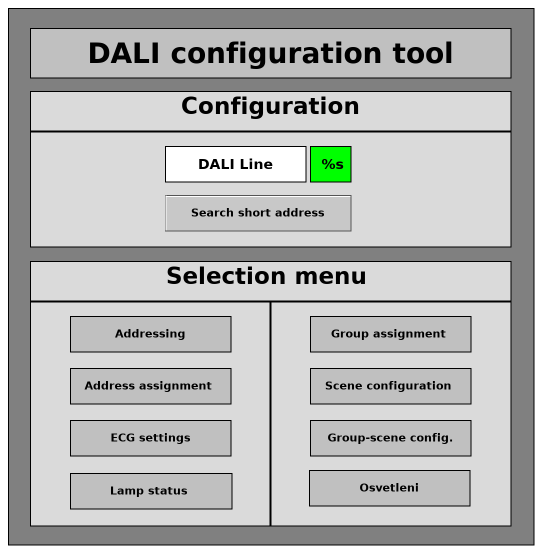
rectangle at (171,91)-(652,247): text "Configuration"
rectangle at (171,261)-(652,526): text "Selection menu"
rectangle at (171,28)-(652,78): text "DALI configuration tool"
rectangle at (211,316)-(372,352): text "Addressing"; opens Addressing
rectangle at (211,368)-(372,404): text "Address assignment"; opens Sort_short_address
rectangle at (451,316)-(612,352): text "Group assignment"; opens group_assignment
rectangle at (451,368)-(612,404): text "Scene configuration"; opens Scene_configuration
rectangle at (211,420)-(372,456): text "ECG settings"; opens ECG_settings
rectangle at (451,420)-(612,456): text "Group-scene config."; opens GroupSceneConfiguration
rectangle at (306,146)-(447,182): text "DALI Line"
button at (306,195)-(492,231): text "Search short address"; taps DALI_Config.SucheKurzadr; tooltip Clicking the button "Search Short Address" will start the search for available short addresses.
rectangle at (451,146)-(492,182): text "%s"; shows DALI_Config.Dali_Linie; alarm colour if DALI_Config.keineJobliste; tooltip Select DALI Line (1 - 5); editable
rectangle at (211,473)-(373,509): text "Lamp status"; opens Lamp_status
rectangle at (450,470)-(611,506): text "Osvetleni"; opens PLC_VISU
4 more shapes without text or variables
*)

(* Visualisation DALI_cfg
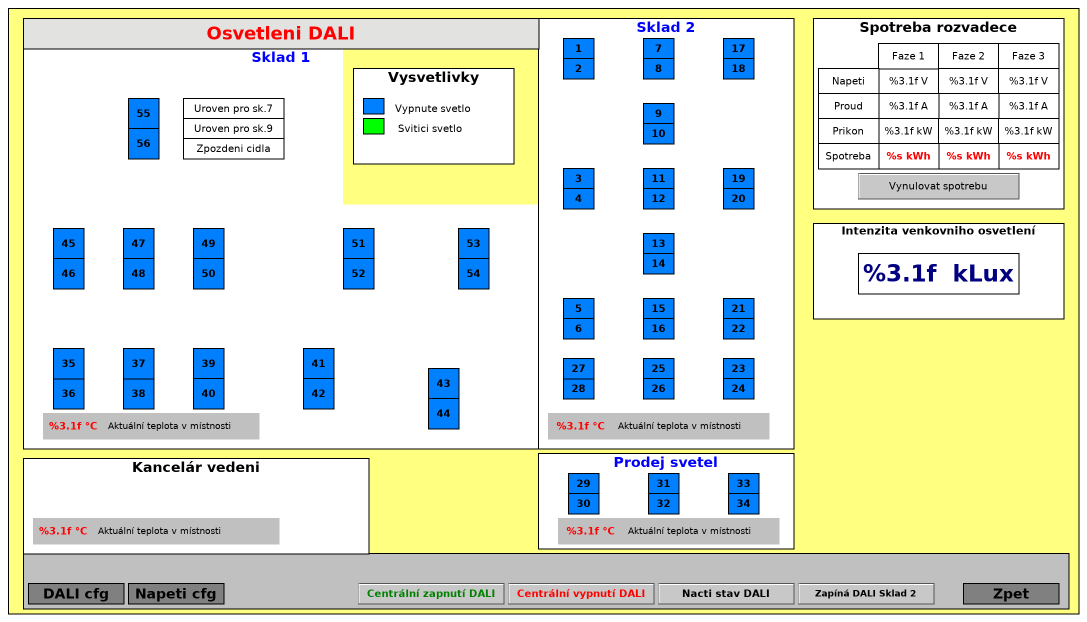
rectangle at (30,50)-(546,451): text "Sklad 1"
rounded rectangle at (360,70)-(521,166): text "Vysvetlivky"
rectangle at (545,455)-(801,551): text "Prodej svetel"; opens prodej_svetel
rectangle at (545,20)-(801,451): text "Sklad 2"; opens prodej_svetel
rectangle at (570,40)-(601,61): text "1"; alarm colour if DALI_Config.Kurzadr[1]
rectangle at (570,40)-(601,61): text "1"; invisible if not DALI_Config.Kurzadr[1]; alarm colour if DALI_Config.LampeEin[1]
rectangle at (570,60)-(601,81): text "2"; alarm colour if DALI_Config.Kurzadr[2]
rectangle at (570,60)-(601,81): text "2"; invisible if not DALI_Config.Kurzadr[2]; alarm colour if DALI_Config.LampeEin[2]
rectangle at (570,170)-(601,191): text "3"; alarm colour if DALI_Config.Kurzadr[3]
rectangle at (570,170)-(601,191): text "3"; invisible if not DALI_Config.Kurzadr[3]; alarm colour if DALI_Config.LampeEin[3]
rectangle at (570,190)-(601,211): text "4"; alarm colour if DALI_Config.Kurzadr[4]
rectangle at (570,190)-(601,211): text "4"; invisible if not DALI_Config.Kurzadr[4]; alarm colour if DALI_Config.LampeEin[4]
rectangle at (570,300)-(601,321): text "5"; alarm colour if DALI_Config.Kurzadr[5]
rectangle at (570,300)-(601,321): text "5"; invisible if not DALI_Config.Kurzadr[5]; alarm colour if DALI_Config.LampeEin[5]
rectangle at (570,320)-(601,341): text "6"; alarm colour if DALI_Config.Kurzadr[6]
rectangle at (570,320)-(601,341): text "6"; invisible if not DALI_Config.Kurzadr[6]; alarm colour if DALI_Config.LampeEin[6]
rectangle at (650,40)-(681,61): text "7"; alarm colour if DALI_Config.Kurzadr[7]
rectangle at (650,40)-(681,61): text "7"; invisible if not DALI_Config.Kurzadr[7]; alarm colour if DALI_Config.LampeEin[7]
rectangle at (650,60)-(681,81): text "8"; alarm colour if DALI_Config.Kurzadr[8]
rectangle at (650,60)-(681,81): text "8"; invisible if not DALI_Config.Kurzadr[8]; alarm colour if DALI_Config.LampeEin[8]
rectangle at (650,105)-(681,126): text "9"; alarm colour if DALI_Config.Kurzadr[9]
rectangle at (650,105)-(681,126): text "9"; invisible if not DALI_Config.Kurzadr[9]; alarm colour if DALI_Config.LampeEin[9]
rectangle at (650,125)-(681,146): text "10"; alarm colour if DALI_Config.Kurzadr[10]
rectangle at (650,125)-(681,146): text "10"; invisible if not DALI_Config.Kurzadr[10]; alarm colour if DALI_Config.LampeEin[10]
rectangle at (650,170)-(681,191): text "11"; alarm colour if DALI_Config.Kurzadr[11]
rectangle at (650,170)-(681,191): text "11"; invisible if not DALI_Config.Kurzadr[11]; alarm colour if DALI_Config.LampeEin[11]
rectangle at (650,190)-(681,211): text "12"; alarm colour if DALI_Config.Kurzadr[12]
rectangle at (650,190)-(681,211): text "12"; invisible if not DALI_Config.Kurzadr[12]; alarm colour if DALI_Config.LampeEin[12]
rectangle at (650,235)-(681,256): text "13"; alarm colour if DALI_Config.Kurzadr[13]
rectangle at (650,235)-(681,256): text "13"; invisible if not DALI_Config.Kurzadr[13]; alarm colour if DALI_Config.LampeEin[13]
rectangle at (650,255)-(681,276): text "14"; alarm colour if DALI_Config.Kurzadr[14]
rectangle at (650,255)-(681,276): text "14"; invisible if not DALI_Config.Kurzadr[14]; alarm colour if DALI_Config.LampeEin[14]
rectangle at (650,300)-(681,321): text "15"; alarm colour if DALI_Config.Kurzadr[15]
rectangle at (650,300)-(681,321): text "15"; invisible if not DALI_Config.Kurzadr[15]; alarm colour if DALI_Config.LampeEin[15]
rectangle at (650,320)-(681,341): text "16"; alarm colour if DALI_Config.Kurzadr[16]
rectangle at (650,320)-(681,341): text "16"; invisible if not DALI_Config.Kurzadr[16]; alarm colour if DALI_Config.LampeEin[16]
rectangle at (730,40)-(761,61): text "17"; alarm colour if DALI_Config.Kurzadr[17]
rectangle at (730,40)-(761,61): text "17"; invisible if not DALI_Config.Kurzadr[17]; alarm colour if DALI_Config.LampeEin[17]
rectangle at (730,170)-(761,191): text "19"; alarm colour if DALI_Config.Kurzadr[19]
rectangle at (730,170)-(761,191): text "19"; invisible if not DALI_Config.Kurzadr[19]; alarm colour if DALI_Config.LampeEin[19]
rectangle at (730,60)-(761,81): text "18"; alarm colour if DALI_Config.Kurzadr[18]
rectangle at (730,60)-(761,81): text "18"; invisible if not DALI_Config.Kurzadr[18]; alarm colour if DALI_Config.LampeEin[18]
rectangle at (730,190)-(761,211): text "20"; alarm colour if DALI_Config.Kurzadr[20]
rectangle at (730,190)-(761,211): text "20"; invisible if not DALI_Config.Kurzadr[20]; alarm colour if DALI_Config.LampeEin[20]
rectangle at (730,300)-(761,321): text "21"; alarm colour if DALI_Config.Kurzadr[21]
rectangle at (730,300)-(761,321): text "21"; invisible if not DALI_Config.Kurzadr[21]; alarm colour if DALI_Config.LampeEin[21]
rectangle at (730,320)-(761,341): text "22"; alarm colour if DALI_Config.Kurzadr[22]
rectangle at (730,320)-(761,341): text "22"; invisible if not DALI_Config.Kurzadr[22]; alarm colour if DALI_Config.LampeEin[22]
rectangle at (730,360)-(761,381): text "23"; alarm colour if DALI_Config.Kurzadr[23]
rectangle at (730,360)-(761,381): text "23"; invisible if not DALI_Config.Kurzadr[23]; alarm colour if DALI_Config.LampeEin[23]
rectangle at (730,380)-(761,401): text "24"; alarm colour if DALI_Config.Kurzadr[24]
rectangle at (730,380)-(761,401): text "24"; invisible if not DALI_Config.Kurzadr[24]; alarm colour if DALI_Config.LampeEin[24]
rectangle at (650,360)-(681,381): text "25"; alarm colour if DALI_Config.Kurzadr[25]
rectangle at (650,360)-(681,381): text "25"; invisible if not DALI_Config.Kurzadr[25]; alarm colour if DALI_Config.LampeEin[25]
rectangle at (575,475)-(606,496): text "29"; alarm colour if DALI_Config.Kurzadr[29]
rectangle at (575,475)-(606,496): text "29"; invisible if not DALI_Config.Kurzadr[29]; alarm colour if DALI_Config.LampeEin[29]
rectangle at (570,380)-(601,401): text "28"; alarm colour if DALI_Config.Kurzadr[28]
rectangle at (570,380)-(601,401): text "28"; invisible if not DALI_Config.Kurzadr[28]; alarm colour if DALI_Config.LampeEin[28]
rectangle at (570,360)-(601,381): text "27"; alarm colour if DALI_Config.Kurzadr[27]
rectangle at (570,360)-(601,381): text "27"; invisible if not DALI_Config.Kurzadr[27]; alarm colour if DALI_Config.LampeEin[27]
rectangle at (650,380)-(681,401): text "26"; alarm colour if DALI_Config.Kurzadr[26]
rectangle at (650,380)-(681,401): text "26"; invisible if not DALI_Config.Kurzadr[26]; alarm colour if DALI_Config.LampeEin[26]
rectangle at (575,495)-(606,516): text "30"; alarm colour if DALI_Config.Kurzadr[30]
rectangle at (575,495)-(606,516): text "30"; invisible if not DALI_Config.Kurzadr[30]; alarm colour if DALI_Config.LampeEin[30]
rectangle at (655,475)-(686,496): text "31"; alarm colour if DALI_Config.Kurzadr[31]
rectangle at (655,475)-(686,496): text "31"; invisible if not DALI_Config.Kurzadr[31]; alarm colour if DALI_Config.LampeEin[31]
rectangle at (655,495)-(686,516): text "32"; alarm colour if DALI_Config.Kurzadr[32]
rectangle at (655,495)-(686,516): text "32"; invisible if not DALI_Config.Kurzadr[32]; alarm colour if DALI_Config.LampeEin[32]
rectangle at (735,475)-(766,496): text "33"; alarm colour if DALI_Config.Kurzadr[33]
rectangle at (735,475)-(766,496): text "33"; invisible if not DALI_Config.Kurzadr[33]; alarm colour if DALI_Config.LampeEin[33]
rectangle at (735,495)-(766,516): text "34"; alarm colour if DALI_Config.Kurzadr[34]
rectangle at (735,495)-(766,516): text "34"; invisible if not DALI_Config.Kurzadr[34]; alarm colour if DALI_Config.LampeEin[34]
rectangle at (60,380)-(91,411): text "36"; alarm colour if DALI_Config.Kurzadr[36]
rectangle at (60,380)-(91,411): text "36"; invisible if not DALI_Config.Kurzadr[36]; alarm colour if DALI_Config.LampeEin[36]
rectangle at (130,380)-(161,411): text "38"; alarm colour if DALI_Config.Kurzadr[38]
rectangle at (130,380)-(161,411): text "38"; invisible if not DALI_Config.Kurzadr[38]; alarm colour if DALI_Config.LampeEin[38]
rectangle at (200,350)-(231,381): text "39"; alarm colour if DALI_Config.Kurzadr[39]
rectangle at (200,350)-(231,381): text "39"; invisible if not DALI_Config.Kurzadr[39]; alarm colour if DALI_Config.LampeEin[39]
rectangle at (130,350)-(161,381): text "37"; alarm colour if DALI_Config.Kurzadr[37]
rectangle at (130,350)-(161,381): text "37"; invisible if not DALI_Config.Kurzadr[37]; alarm colour if DALI_Config.LampeEin[37]
rectangle at (60,350)-(91,381): text "35"; alarm colour if DALI_Config.Kurzadr[35]
rectangle at (60,350)-(91,381): text "35"; invisible if not DALI_Config.Kurzadr[35]; alarm colour if DALI_Config.LampeEin[35]
rectangle at (310,350)-(341,381): text "41"; alarm colour if DALI_Config.Kurzadr[41]
rectangle at (310,350)-(341,381): text "41"; invisible if not DALI_Config.Kurzadr[41]; alarm colour if DALI_Config.LampeEin[41]
rectangle at (310,380)-(341,411): text "42"; alarm colour if DALI_Config.Kurzadr[42]
rectangle at (310,380)-(341,411): text "42"; invisible if not DALI_Config.Kurzadr[42]; alarm colour if DALI_Config.LampeEin[42]
rectangle at (200,380)-(231,411): text "40"; alarm colour if DALI_Config.Kurzadr[40]
rectangle at (200,380)-(231,411): text "40"; invisible if not DALI_Config.Kurzadr[40]; alarm colour if DALI_Config.LampeEin[40]
rectangle at (435,370)-(466,401): text "43"; alarm colour if DALI_Config.Kurzadr[43]
rectangle at (435,370)-(466,401): text "43"; invisible if not DALI_Config.Kurzadr[43]; alarm colour if DALI_Config.LampeEin[43]
rectangle at (435,400)-(466,431): text "44"; alarm colour if DALI_Config.Kurzadr[44]
rectangle at (435,400)-(466,431): text "44"; invisible if not DALI_Config.Kurzadr[44]; alarm colour if DALI_Config.LampeEin[44]
rectangle at (60,230)-(91,261): text "45"; alarm colour if DALI_Config.Kurzadr[45]
rectangle at (60,230)-(91,261): text "45"; invisible if not DALI_Config.Kurzadr[45]; alarm colour if DALI_Config.LampeEin[45]
rectangle at (60,260)-(91,291): text "46"; alarm colour if DALI_Config.Kurzadr[46]
rectangle at (60,260)-(91,291): text "46"; invisible if not DALI_Config.Kurzadr[46]; alarm colour if DALI_Config.LampeEin[46]
rectangle at (130,230)-(161,261): text "47"; alarm colour if DALI_Config.Kurzadr[47]
rectangle at (130,230)-(161,261): text "47"; invisible if not DALI_Config.Kurzadr[47]; alarm colour if DALI_Config.LampeEin[47]
rectangle at (130,260)-(161,291): text "48"; alarm colour if DALI_Config.Kurzadr[48]
rectangle at (130,260)-(161,291): text "48"; invisible if not DALI_Config.Kurzadr[48]; alarm colour if DALI_Config.LampeEin[48]
rectangle at (200,230)-(231,261): text "49"; alarm colour if DALI_Config.Kurzadr[49]
rectangle at (200,230)-(231,261): text "49"; invisible if not DALI_Config.Kurzadr[49]; alarm colour if DALI_Config.LampeEin[49]
rectangle at (200,260)-(231,291): text "50"; alarm colour if DALI_Config.Kurzadr[50]
rectangle at (200,260)-(231,291): text "50"; invisible if not DALI_Config.Kurzadr[50]; alarm colour if DALI_Config.LampeEin[50]
rectangle at (350,230)-(381,261): text "51"; alarm colour if DALI_Config.Kurzadr[51]
rectangle at (350,230)-(381,261): text "51"; invisible if not DALI_Config.Kurzadr[51]; alarm colour if DALI_Config.LampeEin[51]
rectangle at (350,260)-(381,291): text "52"; alarm colour if DALI_Config.Kurzadr[52]
rectangle at (350,260)-(381,291): text "52"; invisible if not DALI_Config.Kurzadr[52]; alarm colour if DALI_Config.LampeEin[52]
rectangle at (465,230)-(496,261): text "53"; alarm colour if DALI_Config.Kurzadr[53]
rectangle at (465,230)-(496,261): text "53"; invisible if not DALI_Config.Kurzadr[53]; alarm colour if DALI_Config.LampeEin[53]
rectangle at (465,260)-(496,291): text "54"; alarm colour if DALI_Config.Kurzadr[54]
rectangle at (465,260)-(496,291): text "54"; invisible if not DALI_Config.Kurzadr[54]; alarm colour if DALI_Config.LampeEin[54]
rectangle at (135,100)-(166,131): text "55"; alarm colour if DALI_Config.Kurzadr[55]
rectangle at (135,100)-(166,131): text "55"; invisible if not DALI_Config.Kurzadr[55]; alarm colour if DALI_Config.LampeEin[55]
rectangle at (135,130)-(166,161): text "56"; alarm colour if DALI_Config.Kurzadr[56]
rectangle at (135,130)-(166,161): text "56"; invisible if not DALI_Config.Kurzadr[56]; alarm colour if DALI_Config.LampeEin[56]
rectangle at (30,20)-(546,51): text "Osvetleni DALI"
button at (665,585)-(801,606): text "Nacti stav DALI"; taps DALI_Config.Status; tooltip Kliknutim nactete status svetel. (sviti, nesviti, vadna).
rectangle at (400,100)-(516,121): text "Vypnute svetlo"
rectangle at (400,120)-(536,141): text "Svitici svetlo"
rectangle at (565,520)-(631,546): text "%3.1f °C"; shows .Teplota_2/10.0
rectangle at (630,520)-(786,546): text "Aktuální teplota v místnosti"
rectangle at (620,415)-(776,441): text "Aktuální teplota v místnosti"
rectangle at (110,415)-(266,441): text "Aktuální teplota v místnosti"
rectangle at (555,415)-(621,441): text "%3.1f °C"; shows .Teplota_1/10.0
rectangle at (50,415)-(111,441): text "%3.1f °C"; shows .Teplota_3/10.0
button at (365,585)-(511,606): text "Centrální zapnutí DALI"; taps DALI_Config.Ein; tooltip Vsechny DALI svetla zapni
button at (515,585)-(661,606): text "Centrální vypnutí DALI"; taps DALI_Config.Aus; tooltip Vsechny DALI svetla vypni
rounded rectangle at (820,20)-(1071,211): text "Spotreba rozvadece"
rectangle at (885,70)-(946,96): text "%3.1f V"; shows TriFaze.arNapeti[1]
rectangle at (885,45)-(946,71): text "Faze 1"
rectangle at (945,45)-(1006,71): text "Faze 2"
rectangle at (1005,45)-(1066,71): text "Faze 3"
rectangle at (945,70)-(1006,96): text "%3.1f V"; shows TriFaze.arNapeti[2]
rectangle at (1005,70)-(1066,96): text "%3.1f V"; shows TriFaze.arNapeti[3]
rectangle at (1005,95)-(1066,121): text "%3.1f A"; shows TriFaze.arProud[3]
rectangle at (945,95)-(1006,121): text "%3.1f A"; shows TriFaze.arProud[2]
rectangle at (885,95)-(946,121): text "%3.1f A"; shows TriFaze.arProud[1]
rectangle at (885,120)-(946,146): text "%3.1f kW"; shows TriFaze.arVykon[1]
rectangle at (945,120)-(1006,146): text "%3.1f kW"; shows TriFaze.arVykon[2]
rectangle at (1005,120)-(1066,146): text "%3.1f kW"; shows TriFaze.arVykon[3]
rectangle at (1005,145)-(1066,171): text "%s kWh"; shows TriFaze.adwSpotreba[3]
rectangle at (945,145)-(1006,171): text "%s kWh"; shows TriFaze.adwSpotreba[2]
rectangle at (885,145)-(946,171): text "%s kWh"; shows TriFaze.adwSpotreba[1]
button at (865,175)-(1026,201): text "Vynulovat spotrebu"; taps TriFaze.SmazL1
rounded rectangle at (820,225)-(1071,321): text "Intenzita venkovniho osvetlení"; opens lux
rectangle at (865,255)-(1026,296): text "%3.1f  kLux"; shows .Analog_1/3276.4*2
rectangle at (825,70)-(886,96): text "Napeti"
rectangle at (825,95)-(886,121): text "Proud"
rectangle at (825,120)-(886,146): text "Prikon"
rectangle at (825,145)-(886,171): text "Spotreba"
rectangle at (30,460)-(376,556): text "Kancelár vedeni"
rectangle at (100,520)-(286,546): text "Aktuální teplota v místnosti"
rectangle at (40,520)-(101,546): text "%3.1f °C"; shows .Teplota_4/10.0
rectangle at (970,585)-(1066,606): text "Zpet"; opens PLC_VISU; tooltip Na úvodní stranu
rectangle at (135,585)-(231,606): text "Napeti cfg"; opens Visualizace; tooltip Back to home page
button at (805,585)-(941,606): text "Zapíná DALI Sklad 2"; taps .TL01s; tooltip 1x zapne/vypne, 2x zapne skupinu 2, 3x zapne vše
rectangle at (35,585)-(131,606): text "DALI cfg"; opens DALI; tooltip Back to home page
rectangle at (190,100)-(291,121): text "Uroven pro sk.7"
rectangle at (190,120)-(291,141): text "Uroven pro sk.9"
rectangle at (190,140)-(291,161): text "Zpozdeni cidla"
6 more shapes without text or variables
3 elements of other kinds (tables, trends, ...) not read
*)

(* Visualisation ECG_settings
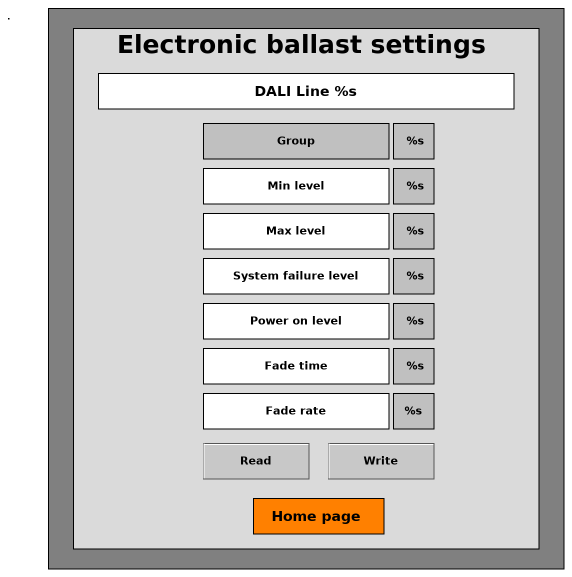
rectangle at (150,40)-(616,561): text "Electronic ballast settings"
rectangle at (280,225)-(466,261): text "Max level"
rectangle at (280,180)-(466,216): text "Min level"
rectangle at (280,270)-(466,306): text "System failure level"
rectangle at (280,315)-(466,351): text "Power on level"
rectangle at (280,360)-(466,396): text "Fade time"
rectangle at (280,405)-(466,441): text "Fade rate"
rectangle at (280,135)-(466,171): text "Short address"; invisible if DALI_Config.Kurzadr_Gruppe; toggles DALI_Config.Kurzadr_Gruppe
rectangle at (280,135)-(466,171): text "Group"; invisible if not DALI_Config.Kurzadr_Gruppe; toggles DALI_Config.Kurzadr_Gruppe; tooltip Selection group or short address
rectangle at (470,135)-(511,171): text "%s"; shows DALI_Config.Adresse; tooltip Enter group (1-16) or short address (1 - 64); editable
rounded rectangle at (330,510)-(461,546): text "Home page"; opens DALI; tooltip Back to home page
rectangle at (470,180)-(511,216): text "%s"; shows DALI_Config.MinLevel; tooltip Minimal brightness level in percent. Min level has to be smaller than max level.; editable
rectangle at (470,225)-(511,261): text "%s"; shows DALI_Config.MaxLevel; tooltip Maximum brightness level in percent; editable
rectangle at (470,270)-(511,306): text "%s"; shows DALI_Config.SystemFailure; tooltip Brightness level in percent in case of a system failure. The value 101 means "MASK".; editable
rectangle at (470,315)-(511,351): text "%s"; shows DALI_Config.PowerOn; tooltip Brightness level in percent if the ECGs are powered on.; editable
rectangle at (470,360)-(511,396): text "%s"; shows DALI_Config.Konfig[4]; tooltip Enter the fade time (0 - 15); editable
rectangle at (470,405)-(511,441): text "%s"; shows DALI_Config.Konfig[5]; tooltip Enter the fade rate (1 -15); editable
button at (280,455)-(386,491): text "Read"; taps DALI_Config.Lese; tooltip If you click the button "Read", the settings of the ECG will be read. Group queries are not possible.
button at (405,455)-(511,491): text "Write"; taps DALI_Config.Schreib; tooltip If you click the button "Write", the new settings will be written into the ECG.
rounded rectangle at (175,85)-(591,121): text "DALI Line %s"; shows DALI_Config.bDali_Linie; tooltip You can change the DALI Line only on the home page.
2 more shapes without text or variables
*)

(* Visualisation Group_assignment
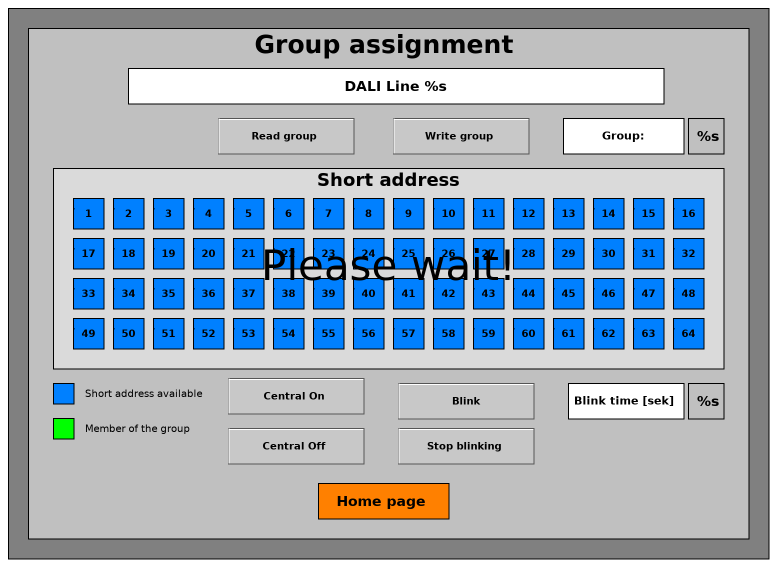
rectangle at (40,40)-(761,551): text "Group assignment"
rounded rectangle at (330,495)-(461,531): text "Home page"; opens DALI; tooltip Back to home page
rectangle at (65,180)-(736,381): text "Short address"
rectangle at (85,210)-(116,241): text "1"; alarm colour if DALI_Config.Kurzadr[1]
rectangle at (85,210)-(116,241): text "1"; invisible if not DALI_Config.Kurzadr[1]; alarm colour if DALI_Config.Gruppenadr[1]; toggles DALI_Config.Gruppenadr[1]
rectangle at (125,210)-(156,241): text "2"; alarm colour if DALI_Config.Kurzadr[2]
rectangle at (125,210)-(156,241): text "2"; invisible if not DALI_Config.Kurzadr[2]; alarm colour if DALI_Config.Gruppenadr[2]; toggles DALI_Config.Gruppenadr[2]
rectangle at (165,210)-(196,241): text "3"; alarm colour if DALI_Config.Kurzadr[3]
rectangle at (165,210)-(196,241): text "3"; invisible if not DALI_Config.Kurzadr[3]; alarm colour if DALI_Config.Gruppenadr[3]; toggles DALI_Config.Gruppenadr[3]
rectangle at (205,210)-(236,241): text "4"; alarm colour if DALI_Config.Kurzadr[4]
rectangle at (205,210)-(236,241): text "4"; invisible if not DALI_Config.Kurzadr[4]; alarm colour if DALI_Config.Gruppenadr[4]; toggles DALI_Config.Gruppenadr[4]
rectangle at (245,210)-(276,241): text "5"; alarm colour if DALI_Config.Kurzadr[5]
rectangle at (245,210)-(276,241): text "5"; invisible if not DALI_Config.Kurzadr[5]; alarm colour if DALI_Config.Gruppenadr[5]; toggles DALI_Config.Gruppenadr[5]
rectangle at (285,210)-(316,241): text "6"; alarm colour if DALI_Config.Kurzadr[6]
rectangle at (285,210)-(316,241): text "6"; invisible if not DALI_Config.Kurzadr[6]; alarm colour if DALI_Config.Gruppenadr[6]; toggles DALI_Config.Gruppenadr[6]
rectangle at (325,210)-(356,241): text "7"; alarm colour if DALI_Config.Kurzadr[7]
rectangle at (325,210)-(356,241): text "7"; invisible if not DALI_Config.Kurzadr[7]; alarm colour if DALI_Config.Gruppenadr[7]; toggles DALI_Config.Gruppenadr[7]
rectangle at (365,210)-(396,241): text "8"; alarm colour if DALI_Config.Kurzadr[8]
rectangle at (365,210)-(396,241): text "8"; invisible if not DALI_Config.Kurzadr[8]; alarm colour if DALI_Config.Gruppenadr[8]; toggles DALI_Config.Gruppenadr[8]
rectangle at (405,210)-(436,241): text "9"; alarm colour if DALI_Config.Kurzadr[9]
rectangle at (405,210)-(436,241): text "9"; invisible if not DALI_Config.Kurzadr[9]; alarm colour if DALI_Config.Gruppenadr[9]; toggles DALI_Config.Gruppenadr[9]
rectangle at (445,210)-(476,241): text "10"; alarm colour if DALI_Config.Kurzadr[10]
rectangle at (445,210)-(476,241): text "10"; invisible if not DALI_Config.Kurzadr[10]; alarm colour if DALI_Config.Gruppenadr[10]; toggles DALI_Config.Gruppenadr[10]
rectangle at (485,210)-(516,241): text "11"; alarm colour if DALI_Config.Kurzadr[11]
rectangle at (485,210)-(516,241): text "11"; invisible if not DALI_Config.Kurzadr[11]; alarm colour if DALI_Config.Gruppenadr[11]; toggles DALI_Config.Gruppenadr[11]
rectangle at (525,210)-(556,241): text "12"; alarm colour if DALI_Config.Kurzadr[12]
rectangle at (525,210)-(556,241): text "12"; invisible if not DALI_Config.Kurzadr[12]; alarm colour if DALI_Config.Gruppenadr[12]; toggles DALI_Config.Gruppenadr[12]
rectangle at (565,210)-(596,241): text "13"; alarm colour if DALI_Config.Kurzadr[13]
rectangle at (565,210)-(596,241): text "13"; invisible if not DALI_Config.Kurzadr[13]; alarm colour if DALI_Config.Gruppenadr[13]; toggles DALI_Config.Gruppenadr[13]
rectangle at (605,210)-(636,241): text "14"; alarm colour if DALI_Config.Kurzadr[14]
rectangle at (605,210)-(636,241): text "14"; invisible if not DALI_Config.Kurzadr[14]; alarm colour if DALI_Config.Gruppenadr[14]; toggles DALI_Config.Gruppenadr[14]
rectangle at (645,210)-(676,241): text "15"; alarm colour if DALI_Config.Kurzadr[15]
rectangle at (645,210)-(676,241): text "15"; invisible if not DALI_Config.Kurzadr[15]; alarm colour if DALI_Config.Gruppenadr[15]; toggles DALI_Config.Gruppenadr[15]
rectangle at (685,210)-(716,241): text "16"; alarm colour if DALI_Config.Kurzadr[16]
rectangle at (685,210)-(716,241): text "16"; invisible if not DALI_Config.Kurzadr[16]; alarm colour if DALI_Config.Gruppenadr[16]; toggles DALI_Config.Gruppenadr[16]
button at (405,130)-(541,166): text "Write group"; taps DALI_Config.Gruppenkonfiguration; tooltip If you click the button "Write Group", the marked short addresses will be saved as a group.
rectangle at (575,130)-(696,166): text "Group:"
rectangle at (700,130)-(736,166): text "%s"; shows DALI_Config.Gruppe; tooltip Enter the number of the group (1 - 16); editable
button at (410,395)-(546,431): text "Blink"; taps DALI_Config.BlinkenGruppe; tooltip If you click the button "Blink", the selected ECG will blink as long as defined by the "Blink Time" parameter.
button at (410,440)-(546,476): text "Stop blinking"; taps DALI_Config.xBlinken_Aus; tooltip If you click the button "Stop blinking", the blinking of the ECG will stop immediately.
button at (230,130)-(366,166): text "Read group"; taps DALI_Config.GruppeLesen; tooltip If you click the button "Read Group", the short addresses that belong to the group will be displayed.
rectangle at (95,395)-(226,416): text "Short address available"
rectangle at (95,430)-(246,451): text "Member of the group"
rounded rectangle at (140,80)-(676,116): text "DALI Line %s"; shows DALI_Config.bDali_Linie; tooltip You can change the DALI Line only on the home page.
rectangle at (85,250)-(116,281): text "17"; alarm colour if DALI_Config.Kurzadr[17]
rectangle at (85,250)-(116,281): text "17"; invisible if not DALI_Config.Kurzadr[17]; alarm colour if DALI_Config.Gruppenadr[17]; toggles DALI_Config.Gruppenadr[17]
rectangle at (125,250)-(156,281): text "18"; alarm colour if DALI_Config.Kurzadr[18]
rectangle at (125,250)-(156,281): text "18"; invisible if not DALI_Config.Kurzadr[18]; alarm colour if DALI_Config.Gruppenadr[18]; toggles DALI_Config.Gruppenadr[18]
rectangle at (165,250)-(196,281): text "19"; alarm colour if DALI_Config.Kurzadr[19]
rectangle at (165,250)-(196,281): text "19"; invisible if not DALI_Config.Kurzadr[19]; alarm colour if DALI_Config.Gruppenadr[19]; toggles DALI_Config.Gruppenadr[19]
rectangle at (205,250)-(236,281): text "20"; alarm colour if DALI_Config.Kurzadr[20]
rectangle at (205,250)-(236,281): text "20"; invisible if not DALI_Config.Kurzadr[20]; alarm colour if DALI_Config.Gruppenadr[20]; toggles DALI_Config.Gruppenadr[20]
rectangle at (245,250)-(276,281): text "21"; alarm colour if DALI_Config.Kurzadr[21]
rectangle at (245,250)-(276,281): text "21"; invisible if not DALI_Config.Kurzadr[21]; alarm colour if DALI_Config.Gruppenadr[21]; toggles DALI_Config.Gruppenadr[21]
rectangle at (285,250)-(316,281): text "22"; alarm colour if DALI_Config.Kurzadr[22]
rectangle at (285,250)-(316,281): text "22"; invisible if not DALI_Config.Kurzadr[22]; alarm colour if DALI_Config.Gruppenadr[22]; toggles DALI_Config.Gruppenadr[22]
rectangle at (325,250)-(356,281): text "23"; alarm colour if DALI_Config.Kurzadr[23]
rectangle at (325,250)-(356,281): text "23"; invisible if not DALI_Config.Kurzadr[23]; alarm colour if DALI_Config.Gruppenadr[23]; toggles DALI_Config.Gruppenadr[23]
rectangle at (365,250)-(396,281): text "24"; alarm colour if DALI_Config.Kurzadr[24]
rectangle at (365,250)-(396,281): text "24"; invisible if not DALI_Config.Kurzadr[24]; alarm colour if DALI_Config.Gruppenadr[24]; toggles DALI_Config.Gruppenadr[24]
rectangle at (405,250)-(436,281): text "25"; alarm colour if DALI_Config.Kurzadr[25]
rectangle at (405,250)-(436,281): text "25"; invisible if not DALI_Config.Kurzadr[25]; alarm colour if DALI_Config.Gruppenadr[25]; toggles DALI_Config.Gruppenadr[25]
rectangle at (445,250)-(476,281): text "26"; alarm colour if DALI_Config.Kurzadr[26]
rectangle at (445,250)-(476,281): text "26"; invisible if not DALI_Config.Kurzadr[26]; alarm colour if DALI_Config.Gruppenadr[26]; toggles DALI_Config.Gruppenadr[26]
rectangle at (485,250)-(516,281): text "27"; alarm colour if DALI_Config.Kurzadr[27]
rectangle at (485,250)-(516,281): text "27"; invisible if not DALI_Config.Kurzadr[27]; alarm colour if DALI_Config.Gruppenadr[27]; toggles DALI_Config.Gruppenadr[27]
rectangle at (525,250)-(556,281): text "28"; alarm colour if DALI_Config.Kurzadr[28]
rectangle at (525,250)-(556,281): text "28"; invisible if not DALI_Config.Kurzadr[28]; alarm colour if DALI_Config.Gruppenadr[28]; toggles DALI_Config.Gruppenadr[28]
rectangle at (565,250)-(596,281): text "29"; alarm colour if DALI_Config.Kurzadr[29]
rectangle at (565,250)-(596,281): text "29"; invisible if not DALI_Config.Kurzadr[29]; alarm colour if DALI_Config.Gruppenadr[29]; toggles DALI_Config.Gruppenadr[29]
rectangle at (605,250)-(636,281): text "30"; alarm colour if DALI_Config.Kurzadr[30]
rectangle at (605,250)-(636,281): text "30"; invisible if not DALI_Config.Kurzadr[30]; alarm colour if DALI_Config.Gruppenadr[30]; toggles DALI_Config.Gruppenadr[30]
rectangle at (645,250)-(676,281): text "31"; alarm colour if DALI_Config.Kurzadr[31]
rectangle at (645,250)-(676,281): text "31"; invisible if not DALI_Config.Kurzadr[31]; alarm colour if DALI_Config.Gruppenadr[31]; toggles DALI_Config.Gruppenadr[31]
rectangle at (685,250)-(716,281): text "32"; alarm colour if DALI_Config.Kurzadr[32]
rectangle at (685,250)-(716,281): text "32"; invisible if not DALI_Config.Kurzadr[32]; alarm colour if DALI_Config.Gruppenadr[32]; toggles DALI_Config.Gruppenadr[32]
rectangle at (85,290)-(116,321): text "33"; alarm colour if DALI_Config.Kurzadr[33]
rectangle at (85,290)-(116,321): text "33"; invisible if not DALI_Config.Kurzadr[33]; alarm colour if DALI_Config.Gruppenadr[33]; toggles DALI_Config.Gruppenadr[33]
rectangle at (125,290)-(156,321): text "34"; alarm colour if DALI_Config.Kurzadr[34]
rectangle at (125,290)-(156,321): text "34"; invisible if not DALI_Config.Kurzadr[34]; alarm colour if DALI_Config.Gruppenadr[34]; toggles DALI_Config.Gruppenadr[34]
rectangle at (165,290)-(196,321): text "35"; alarm colour if DALI_Config.Kurzadr[35]
rectangle at (165,290)-(196,321): text "35"; invisible if not DALI_Config.Kurzadr[35]; alarm colour if DALI_Config.Gruppenadr[35]; toggles DALI_Config.Gruppenadr[35]
rectangle at (205,290)-(236,321): text "36"; alarm colour if DALI_Config.Kurzadr[36]
rectangle at (205,290)-(236,321): text "36"; invisible if not DALI_Config.Kurzadr[36]; alarm colour if DALI_Config.Gruppenadr[36]; toggles DALI_Config.Gruppenadr[36]
rectangle at (245,290)-(276,321): text "37"; alarm colour if DALI_Config.Kurzadr[37]
rectangle at (245,290)-(276,321): text "37"; invisible if not DALI_Config.Kurzadr[37]; alarm colour if DALI_Config.Gruppenadr[37]; toggles DALI_Config.Gruppenadr[37]
rectangle at (285,290)-(316,321): text "38"; alarm colour if DALI_Config.Kurzadr[38]
rectangle at (285,290)-(316,321): text "38"; invisible if not DALI_Config.Kurzadr[38]; alarm colour if DALI_Config.Gruppenadr[38]; toggles DALI_Config.Gruppenadr[38]
rectangle at (325,290)-(356,321): text "39"; alarm colour if DALI_Config.Kurzadr[39]
rectangle at (325,290)-(356,321): text "39"; invisible if not DALI_Config.Kurzadr[39]; alarm colour if DALI_Config.Gruppenadr[39]; toggles DALI_Config.Gruppenadr[39]
rectangle at (365,290)-(396,321): text "40"; alarm colour if DALI_Config.Kurzadr[40]
rectangle at (365,290)-(396,321): text "40"; invisible if not DALI_Config.Kurzadr[40]; alarm colour if DALI_Config.Gruppenadr[40]; toggles DALI_Config.Gruppenadr[40]
rectangle at (405,290)-(436,321): text "41"; alarm colour if DALI_Config.Kurzadr[41]
rectangle at (405,290)-(436,321): text "41"; invisible if not DALI_Config.Kurzadr[41]; alarm colour if DALI_Config.Gruppenadr[41]; toggles DALI_Config.Gruppenadr[41]
rectangle at (445,290)-(476,321): text "42"; alarm colour if DALI_Config.Kurzadr[42]
rectangle at (445,290)-(476,321): text "42"; invisible if not DALI_Config.Kurzadr[42]; alarm colour if DALI_Config.Gruppenadr[42]; toggles DALI_Config.Gruppenadr[42]
rectangle at (485,290)-(516,321): text "43"; alarm colour if DALI_Config.Kurzadr[43]
rectangle at (485,290)-(516,321): text "43"; invisible if not DALI_Config.Kurzadr[43]; alarm colour if DALI_Config.Gruppenadr[43]; toggles DALI_Config.Gruppenadr[43]
rectangle at (525,290)-(556,321): text "44"; alarm colour if DALI_Config.Kurzadr[44]
rectangle at (525,290)-(556,321): text "44"; invisible if not DALI_Config.Kurzadr[44]; alarm colour if DALI_Config.Gruppenadr[44]; toggles DALI_Config.Gruppenadr[44]
rectangle at (565,290)-(596,321): text "45"; alarm colour if DALI_Config.Kurzadr[45]
rectangle at (565,290)-(596,321): text "45"; invisible if not DALI_Config.Kurzadr[45]; alarm colour if DALI_Config.Gruppenadr[45]; toggles DALI_Config.Gruppenadr[45]
rectangle at (605,290)-(636,321): text "46"; alarm colour if DALI_Config.Kurzadr[46]
rectangle at (605,290)-(636,321): text "46"; invisible if not DALI_Config.Kurzadr[46]; alarm colour if DALI_Config.Gruppenadr[46]; toggles DALI_Config.Gruppenadr[46]
rectangle at (645,290)-(676,321): text "47"; alarm colour if DALI_Config.Kurzadr[47]
rectangle at (645,290)-(676,321): text "47"; invisible if not DALI_Config.Kurzadr[47]; alarm colour if DALI_Config.Gruppenadr[47]; toggles DALI_Config.Gruppenadr[47]
rectangle at (685,290)-(716,321): text "48"; alarm colour if DALI_Config.Kurzadr[48]
rectangle at (685,290)-(716,321): text "48"; invisible if not DALI_Config.Kurzadr[48]; alarm colour if DALI_Config.Gruppenadr[48]; toggles DALI_Config.Gruppenadr[48]
rectangle at (85,330)-(116,361): text "49"; alarm colour if DALI_Config.Kurzadr[49]
rectangle at (85,330)-(116,361): text "49"; invisible if not DALI_Config.Kurzadr[49]; alarm colour if DALI_Config.Gruppenadr[49]; toggles DALI_Config.Gruppenadr[49]
rectangle at (125,330)-(156,361): text "50"; alarm colour if DALI_Config.Kurzadr[50]
rectangle at (125,330)-(156,361): text "50"; invisible if not DALI_Config.Kurzadr[50]; alarm colour if DALI_Config.Gruppenadr[50]; toggles DALI_Config.Gruppenadr[50]
rectangle at (165,330)-(196,361): text "51"; alarm colour if DALI_Config.Kurzadr[51]
rectangle at (165,330)-(196,361): text "51"; invisible if not DALI_Config.Kurzadr[51]; alarm colour if DALI_Config.Gruppenadr[51]; toggles DALI_Config.Gruppenadr[51]
rectangle at (205,330)-(236,361): text "52"; alarm colour if DALI_Config.Kurzadr[52]
rectangle at (205,330)-(236,361): text "52"; invisible if not DALI_Config.Kurzadr[52]; alarm colour if DALI_Config.Gruppenadr[52]; toggles DALI_Config.Gruppenadr[52]
rectangle at (245,330)-(276,361): text "53"; alarm colour if DALI_Config.Kurzadr[53]
rectangle at (245,330)-(276,361): text "53"; invisible if not DALI_Config.Kurzadr[53]; alarm colour if DALI_Config.Gruppenadr[53]; toggles DALI_Config.Gruppenadr[53]
rectangle at (285,330)-(316,361): text "54"; alarm colour if DALI_Config.Kurzadr[54]
rectangle at (285,330)-(316,361): text "54"; invisible if not DALI_Config.Kurzadr[54]; alarm colour if DALI_Config.Gruppenadr[54]; toggles DALI_Config.Gruppenadr[54]
rectangle at (325,330)-(356,361): text "55"; alarm colour if DALI_Config.Kurzadr[55]
rectangle at (325,330)-(356,361): text "55"; invisible if not DALI_Config.Kurzadr[55]; alarm colour if DALI_Config.Gruppenadr[55]; toggles DALI_Config.Gruppenadr[55]
rectangle at (365,330)-(396,361): text "56"; alarm colour if DALI_Config.Kurzadr[56]
rectangle at (365,330)-(396,361): text "56"; invisible if not DALI_Config.Kurzadr[56]; alarm colour if DALI_Config.Gruppenadr[56]; toggles DALI_Config.Gruppenadr[56]
rectangle at (405,330)-(436,361): text "57"; alarm colour if DALI_Config.Kurzadr[57]
rectangle at (405,330)-(436,361): text "57"; invisible if not DALI_Config.Kurzadr[57]; alarm colour if DALI_Config.Gruppenadr[57]; toggles DALI_Config.Gruppenadr[57]
rectangle at (445,330)-(476,361): text "58"; alarm colour if DALI_Config.Kurzadr[58]
rectangle at (445,330)-(476,361): text "58"; invisible if not DALI_Config.Kurzadr[58]; alarm colour if DALI_Config.Gruppenadr[58]; toggles DALI_Config.Gruppenadr[58]
rectangle at (485,330)-(516,361): text "59"; alarm colour if DALI_Config.Kurzadr[59]
rectangle at (485,330)-(516,361): text "59"; invisible if not DALI_Config.Kurzadr[59]; alarm colour if DALI_Config.Gruppenadr[59]; toggles DALI_Config.Gruppenadr[59]
rectangle at (525,330)-(556,361): text "60"; alarm colour if DALI_Config.Kurzadr[60]
rectangle at (525,330)-(556,361): text "60"; invisible if not DALI_Config.Kurzadr[60]; alarm colour if DALI_Config.Gruppenadr[60]; toggles DALI_Config.Gruppenadr[60]
rectangle at (565,330)-(596,361): text "61"; alarm colour if DALI_Config.Kurzadr[61]
rectangle at (565,330)-(596,361): text "61"; invisible if not DALI_Config.Kurzadr[61]; alarm colour if DALI_Config.Gruppenadr[61]; toggles DALI_Config.Gruppenadr[61]
rectangle at (605,330)-(636,361): text "62"; alarm colour if DALI_Config.Kurzadr[62]
rectangle at (605,330)-(636,361): text "62"; invisible if not DALI_Config.Kurzadr[62]; alarm colour if DALI_Config.Gruppenadr[62]; toggles DALI_Config.Gruppenadr[62]
rectangle at (645,330)-(676,361): text "63"; alarm colour if DALI_Config.Kurzadr[63]
rectangle at (645,330)-(676,361): text "63"; invisible if not DALI_Config.Kurzadr[63]; alarm colour if DALI_Config.Gruppenadr[63]; toggles DALI_Config.Gruppenadr[63]
rectangle at (685,330)-(716,361): text "64"; alarm colour if DALI_Config.Kurzadr[64]
rectangle at (685,330)-(716,361): text "64"; invisible if not DALI_Config.Kurzadr[64]; alarm colour if DALI_Config.Gruppenadr[64]; toggles DALI_Config.Gruppenadr[64]
rectangle at (580,395)-(696,431): text "Blink time [sek]"
button at (240,440)-(376,476): text "Central Off"; taps DALI_Config.Aus; tooltip If you click the button "Central Off", all lamps in the network will be switched off.
button at (240,390)-(376,426): text "Central On"; taps DALI_Config.Ein; tooltip If you click the button "Central On", all lamps in the network will be switched on.
rectangle at (700,395)-(736,431): text "%s"; shows DALI_Config.bBlinkzeit; tooltip Enter blink time (3 - 255 seconds); editable
rectangle at (40,80)-(761,474): text "Please wait!"; invisible if NOT DALI_Config.Unsichtbar
67 more shapes without text or variables
*)

(* Visualisation GroupSceneConfiguration
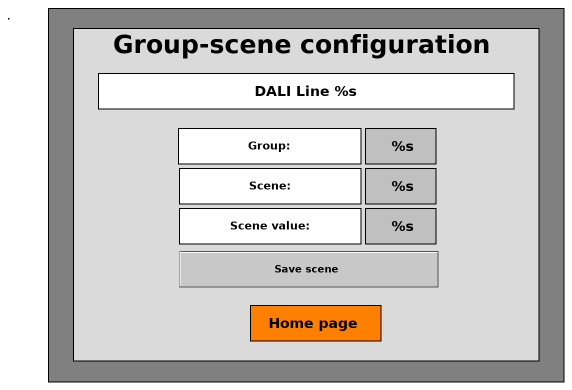
rectangle at (150,40)-(616,373): text "Group-scene configuration"
rounded rectangle at (327,317)-(458,353): text "Home page"; opens DALI; tooltip Back to home page
rounded rectangle at (175,85)-(591,121): text "DALI Line %s"; shows DALI_Config.bDali_Linie; tooltip You can change the DALI Line only on the home page.
rectangle at (255,140)-(438,176): text "Group:"
rectangle at (442,140)-(513,176): text "%s"; shows DALI_Config.sGroup; tooltip Enter the number of the group (1 - 16); editable
button at (256,263)-(515,299): text "Save scene"; taps DALI_Config.sSaveScene; tooltip Save the configured dim levels in the ECGs.
rectangle at (256,180)-(438,216): text "Scene:"
rectangle at (442,180)-(513,216): text "%s"; shows DALI_Config.sScene; tooltip Select scene 1 - 16; editable
rectangle at (256,220)-(438,256): text "Scene value:"
rectangle at (442,220)-(513,256): text "%s"; shows DALI_Config.sSceneValue; tooltip Select scene 1 - 16; editable
2 more shapes without text or variables
*)

(* Visualisation Lamp_status
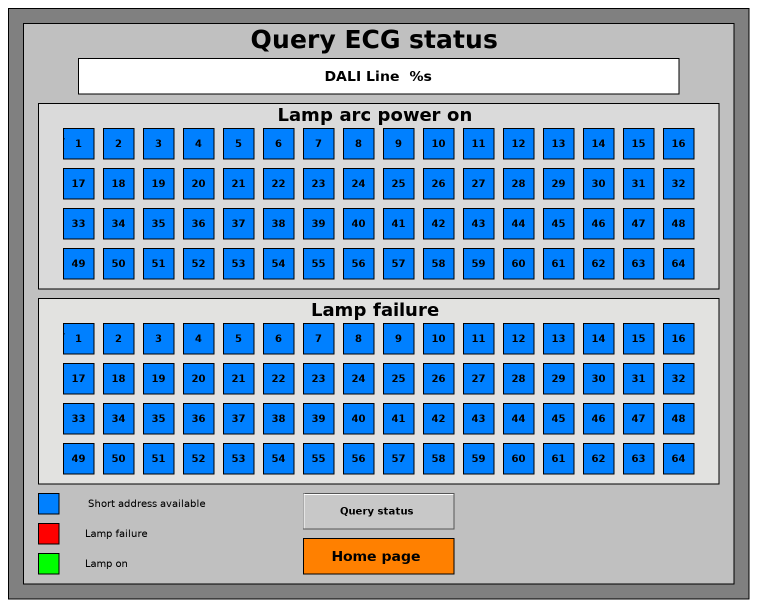
rectangle at (65,35)-(776,596): text "Query ECG status"
rounded rectangle at (345,550)-(496,586): text "Home page"; opens PLC_VISU; tooltip Back to home page
rounded rectangle at (120,70)-(721,106): text "DALI Line  %s"; shows DALI_Config.bDali_Linie; tooltip You can change the DALI Line only on the home page.
rectangle at (80,115)-(761,301): text "Lamp arc power on"
rectangle at (105,140)-(136,171): text "1"; alarm colour if DALI_Config.Kurzadr[1]
rectangle at (105,140)-(136,171): text "1"; invisible if not DALI_Config.Kurzadr[1]; alarm colour if DALI_Config.LampeEin[1]
rectangle at (145,140)-(176,171): text "2"; alarm colour if DALI_Config.Kurzadr[2]
rectangle at (145,140)-(176,171): text "2"; invisible if not DALI_Config.Kurzadr[2]; alarm colour if DALI_Config.LampeEin[2]
rectangle at (185,140)-(216,171): text "3"; alarm colour if DALI_Config.Kurzadr[3]
rectangle at (185,140)-(216,171): text "3"; invisible if not DALI_Config.Kurzadr[3]; alarm colour if DALI_Config.LampeEin[3]
rectangle at (225,140)-(256,171): text "4"; alarm colour if DALI_Config.Kurzadr[4]
rectangle at (225,140)-(256,171): text "4"; invisible if not DALI_Config.Kurzadr[4]; alarm colour if DALI_Config.LampeEin[4]
rectangle at (265,140)-(296,171): text "5"; alarm colour if DALI_Config.Kurzadr[5]
rectangle at (265,140)-(296,171): text "5"; invisible if not DALI_Config.Kurzadr[5]; alarm colour if DALI_Config.LampeEin[5]
rectangle at (305,140)-(336,171): text "6"; alarm colour if DALI_Config.Kurzadr[6]
rectangle at (305,140)-(336,171): text "6"; invisible if not DALI_Config.Kurzadr[6]; alarm colour if DALI_Config.LampeEin[6]
rectangle at (345,140)-(376,171): text "7"; alarm colour if DALI_Config.Kurzadr[7]
rectangle at (345,140)-(376,171): text "7"; invisible if not DALI_Config.Kurzadr[7]; alarm colour if DALI_Config.LampeEin[7]
rectangle at (385,140)-(416,171): text "8"; alarm colour if DALI_Config.Kurzadr[8]
rectangle at (385,140)-(416,171): text "8"; invisible if not DALI_Config.Kurzadr[8]; alarm colour if DALI_Config.LampeEin[8]
rectangle at (425,140)-(456,171): text "9"; alarm colour if DALI_Config.Kurzadr[9]
rectangle at (425,140)-(456,171): text "9"; invisible if not DALI_Config.Kurzadr[9]; alarm colour if DALI_Config.LampeEin[9]
rectangle at (465,140)-(496,171): text "10"; alarm colour if DALI_Config.Kurzadr[10]
rectangle at (465,140)-(496,171): text "10"; invisible if not DALI_Config.Kurzadr[10]; alarm colour if DALI_Config.LampeEin[10]
rectangle at (505,140)-(536,171): text "11"; alarm colour if DALI_Config.Kurzadr[11]
rectangle at (505,140)-(536,171): text "11"; invisible if not DALI_Config.Kurzadr[11]; alarm colour if DALI_Config.LampeEin[11]
rectangle at (545,140)-(576,171): text "12"; alarm colour if DALI_Config.Kurzadr[12]
rectangle at (545,140)-(576,171): text "12"; invisible if not DALI_Config.Kurzadr[12]; alarm colour if DALI_Config.LampeEin[12]
rectangle at (585,140)-(616,171): text "13"; alarm colour if DALI_Config.Kurzadr[13]
rectangle at (585,140)-(616,171): text "13"; invisible if not DALI_Config.Kurzadr[13]; alarm colour if DALI_Config.LampeEin[13]
rectangle at (625,140)-(656,171): text "14"; alarm colour if DALI_Config.Kurzadr[14]
rectangle at (625,140)-(656,171): text "14"; invisible if not DALI_Config.Kurzadr[14]; alarm colour if DALI_Config.LampeEin[14]
rectangle at (665,140)-(696,171): text "15"; alarm colour if DALI_Config.Kurzadr[15]
rectangle at (665,140)-(696,171): text "15"; invisible if not DALI_Config.Kurzadr[15]; alarm colour if DALI_Config.LampeEin[15]
rectangle at (705,140)-(736,171): text "16"; alarm colour if DALI_Config.Kurzadr[16]
rectangle at (705,140)-(736,171): text "16"; invisible if not DALI_Config.Kurzadr[16]; alarm colour if DALI_Config.LampeEin[16]
rectangle at (105,180)-(136,211): text "17"; alarm colour if DALI_Config.Kurzadr[17]
rectangle at (105,180)-(136,211): text "17"; invisible if not DALI_Config.Kurzadr[17]; alarm colour if DALI_Config.LampeEin[17]
rectangle at (185,180)-(216,211): text "19"; alarm colour if DALI_Config.Kurzadr[19]
rectangle at (185,180)-(216,211): text "19"; invisible if not DALI_Config.Kurzadr[19]; alarm colour if DALI_Config.LampeEin[19]
rectangle at (145,180)-(176,211): text "18"; alarm colour if DALI_Config.Kurzadr[18]
rectangle at (145,180)-(176,211): text "18"; invisible if not DALI_Config.Kurzadr[18]; alarm colour if DALI_Config.LampeEin[18]
rectangle at (225,180)-(256,211): text "20"; alarm colour if DALI_Config.Kurzadr[20]
rectangle at (225,180)-(256,211): text "20"; invisible if not DALI_Config.Kurzadr[20]; alarm colour if DALI_Config.LampeEin[20]
rectangle at (265,180)-(296,211): text "21"; alarm colour if DALI_Config.Kurzadr[21]
rectangle at (265,180)-(296,211): text "21"; invisible if not DALI_Config.Kurzadr[21]; alarm colour if DALI_Config.LampeEin[21]
rectangle at (305,180)-(336,211): text "22"; alarm colour if DALI_Config.Kurzadr[22]
rectangle at (305,180)-(336,211): text "22"; invisible if not DALI_Config.Kurzadr[22]; alarm colour if DALI_Config.LampeEin[22]
rectangle at (345,180)-(376,211): text "23"; alarm colour if DALI_Config.Kurzadr[23]
rectangle at (345,180)-(376,211): text "23"; invisible if not DALI_Config.Kurzadr[23]; alarm colour if DALI_Config.LampeEin[23]
rectangle at (385,180)-(416,211): text "24"; alarm colour if DALI_Config.Kurzadr[24]
rectangle at (385,180)-(416,211): text "24"; invisible if not DALI_Config.Kurzadr[24]; alarm colour if DALI_Config.LampeEin[24]
rectangle at (425,180)-(456,211): text "25"; alarm colour if DALI_Config.Kurzadr[25]
rectangle at (425,180)-(456,211): text "25"; invisible if not DALI_Config.Kurzadr[25]; alarm colour if DALI_Config.LampeEin[25]
rectangle at (585,180)-(616,211): text "29"; alarm colour if DALI_Config.Kurzadr[29]
rectangle at (585,180)-(616,211): text "29"; invisible if not DALI_Config.Kurzadr[29]; alarm colour if DALI_Config.LampeEin[29]
rectangle at (545,180)-(576,211): text "28"; alarm colour if DALI_Config.Kurzadr[28]
rectangle at (545,180)-(576,211): text "28"; invisible if not DALI_Config.Kurzadr[28]; alarm colour if DALI_Config.LampeEin[28]
rectangle at (505,180)-(536,211): text "27"; alarm colour if DALI_Config.Kurzadr[27]
rectangle at (505,180)-(536,211): text "27"; invisible if not DALI_Config.Kurzadr[27]; alarm colour if DALI_Config.LampeEin[27]
rectangle at (465,180)-(496,211): text "26"; alarm colour if DALI_Config.Kurzadr[26]
rectangle at (465,180)-(496,211): text "26"; invisible if not DALI_Config.Kurzadr[26]; alarm colour if DALI_Config.LampeEin[26]
rectangle at (625,180)-(656,211): text "30"; alarm colour if DALI_Config.Kurzadr[30]
rectangle at (625,180)-(656,211): text "30"; invisible if not DALI_Config.Kurzadr[30]; alarm colour if DALI_Config.LampeEin[30]
rectangle at (665,180)-(696,211): text "31"; alarm colour if DALI_Config.Kurzadr[31]
rectangle at (665,180)-(696,211): text "31"; invisible if not DALI_Config.Kurzadr[31]; alarm colour if DALI_Config.LampeEin[31]
rectangle at (705,180)-(736,211): text "32"; alarm colour if DALI_Config.Kurzadr[32]
rectangle at (705,180)-(736,211): text "32"; invisible if not DALI_Config.Kurzadr[32]; alarm colour if DALI_Config.LampeEin[32]
rectangle at (105,220)-(136,251): text "33"; alarm colour if DALI_Config.Kurzadr[33]
rectangle at (105,220)-(136,251): text "33"; invisible if not DALI_Config.Kurzadr[33]; alarm colour if DALI_Config.LampeEin[33]
rectangle at (145,220)-(176,251): text "34"; alarm colour if DALI_Config.Kurzadr[34]
rectangle at (145,220)-(176,251): text "34"; invisible if not DALI_Config.Kurzadr[34]; alarm colour if DALI_Config.LampeEin[34]
rectangle at (225,220)-(256,251): text "36"; alarm colour if DALI_Config.Kurzadr[36]
rectangle at (225,220)-(256,251): text "36"; invisible if not DALI_Config.Kurzadr[36]; alarm colour if DALI_Config.LampeEin[36]
rectangle at (305,220)-(336,251): text "38"; alarm colour if DALI_Config.Kurzadr[38]
rectangle at (305,220)-(336,251): text "38"; invisible if not DALI_Config.Kurzadr[38]; alarm colour if DALI_Config.LampeEin[38]
rectangle at (345,220)-(376,251): text "39"; alarm colour if DALI_Config.Kurzadr[39]
rectangle at (345,220)-(376,251): text "39"; invisible if not DALI_Config.Kurzadr[39]; alarm colour if DALI_Config.LampeEin[39]
rectangle at (265,220)-(296,251): text "37"; alarm colour if DALI_Config.Kurzadr[37]
rectangle at (265,220)-(296,251): text "37"; invisible if not DALI_Config.Kurzadr[37]; alarm colour if DALI_Config.LampeEin[37]
rectangle at (185,220)-(216,251): text "35"; alarm colour if DALI_Config.Kurzadr[35]
rectangle at (185,220)-(216,251): text "35"; invisible if not DALI_Config.Kurzadr[35]; alarm colour if DALI_Config.LampeEin[35]
rectangle at (425,220)-(456,251): text "41"; alarm colour if DALI_Config.Kurzadr[41]
rectangle at (425,220)-(456,251): text "41"; invisible if not DALI_Config.Kurzadr[41]; alarm colour if DALI_Config.LampeEin[41]
rectangle at (465,220)-(496,251): text "42"; alarm colour if DALI_Config.Kurzadr[42]
rectangle at (465,220)-(496,251): text "42"; invisible if not DALI_Config.Kurzadr[42]; alarm colour if DALI_Config.LampeEin[42]
rectangle at (385,220)-(416,251): text "40"; alarm colour if DALI_Config.Kurzadr[40]
rectangle at (385,220)-(416,251): text "40"; invisible if not DALI_Config.Kurzadr[40]; alarm colour if DALI_Config.LampeEin[40]
rectangle at (505,220)-(536,251): text "43"; alarm colour if DALI_Config.Kurzadr[43]
rectangle at (505,220)-(536,251): text "43"; invisible if not DALI_Config.Kurzadr[43]; alarm colour if DALI_Config.LampeEin[43]
rectangle at (545,220)-(576,251): text "44"; alarm colour if DALI_Config.Kurzadr[44]
rectangle at (545,220)-(576,251): text "44"; invisible if not DALI_Config.Kurzadr[44]; alarm colour if DALI_Config.LampeEin[44]
rectangle at (585,220)-(616,251): text "45"; alarm colour if DALI_Config.Kurzadr[45]
rectangle at (585,220)-(616,251): text "45"; invisible if not DALI_Config.Kurzadr[45]; alarm colour if DALI_Config.LampeEin[45]
rectangle at (625,220)-(656,251): text "46"; alarm colour if DALI_Config.Kurzadr[46]
rectangle at (625,220)-(656,251): text "46"; invisible if not DALI_Config.Kurzadr[46]; alarm colour if DALI_Config.LampeEin[46]
rectangle at (665,220)-(696,251): text "47"; alarm colour if DALI_Config.Kurzadr[47]
rectangle at (665,220)-(696,251): text "47"; invisible if not DALI_Config.Kurzadr[47]; alarm colour if DALI_Config.LampeEin[47]
rectangle at (705,220)-(736,251): text "48"; alarm colour if DALI_Config.Kurzadr[48]
rectangle at (705,220)-(736,251): text "48"; invisible if not DALI_Config.Kurzadr[48]; alarm colour if DALI_Config.LampeEin[48]
rectangle at (105,260)-(136,291): text "49"; alarm colour if DALI_Config.Kurzadr[49]
rectangle at (105,260)-(136,291): text "49"; invisible if not DALI_Config.Kurzadr[49]; alarm colour if DALI_Config.LampeEin[49]
rectangle at (145,260)-(176,291): text "50"; alarm colour if DALI_Config.Kurzadr[50]
rectangle at (145,260)-(176,291): text "50"; invisible if not DALI_Config.Kurzadr[50]; alarm colour if DALI_Config.LampeEin[50]
rectangle at (185,260)-(216,291): text "51"; alarm colour if DALI_Config.Kurzadr[51]
rectangle at (185,260)-(216,291): text "51"; invisible if not DALI_Config.Kurzadr[51]; alarm colour if DALI_Config.LampeEin[51]
rectangle at (225,260)-(256,291): text "52"; alarm colour if DALI_Config.Kurzadr[52]
rectangle at (225,260)-(256,291): text "52"; invisible if not DALI_Config.Kurzadr[52]; alarm colour if DALI_Config.LampeEin[52]
rectangle at (265,260)-(296,291): text "53"; alarm colour if DALI_Config.Kurzadr[53]
rectangle at (265,260)-(296,291): text "53"; invisible if not DALI_Config.Kurzadr[53]; alarm colour if DALI_Config.LampeEin[53]
rectangle at (305,260)-(336,291): text "54"; alarm colour if DALI_Config.Kurzadr[54]
rectangle at (305,260)-(336,291): text "54"; invisible if not DALI_Config.Kurzadr[54]; alarm colour if DALI_Config.LampeEin[54]
rectangle at (345,260)-(376,291): text "55"; alarm colour if DALI_Config.Kurzadr[55]
rectangle at (345,260)-(376,291): text "55"; invisible if not DALI_Config.Kurzadr[55]; alarm colour if DALI_Config.LampeEin[55]
rectangle at (385,260)-(416,291): text "56"; alarm colour if DALI_Config.Kurzadr[56]
rectangle at (385,260)-(416,291): text "56"; invisible if not DALI_Config.Kurzadr[56]; alarm colour if DALI_Config.LampeEin[56]
rectangle at (425,260)-(456,291): text "57"; alarm colour if DALI_Config.Kurzadr[57]
rectangle at (425,260)-(456,291): text "57"; invisible if not DALI_Config.Kurzadr[57]; alarm colour if DALI_Config.LampeEin[57]
rectangle at (505,260)-(536,291): text "59"; alarm colour if DALI_Config.Kurzadr[59]
rectangle at (505,260)-(536,291): text "59"; invisible if not DALI_Config.Kurzadr[59]; alarm colour if DALI_Config.LampeEin[59]
rectangle at (545,260)-(576,291): text "60"; alarm colour if DALI_Config.Kurzadr[60]
rectangle at (545,260)-(576,291): text "60"; invisible if not DALI_Config.Kurzadr[60]; alarm colour if DALI_Config.LampeEin[60]
rectangle at (585,260)-(616,291): text "61"; alarm colour if DALI_Config.Kurzadr[61]
rectangle at (585,260)-(616,291): text "61"; invisible if not DALI_Config.Kurzadr[61]; alarm colour if DALI_Config.LampeEin[61]
rectangle at (625,260)-(656,291): text "62"; alarm colour if DALI_Config.Kurzadr[62]
rectangle at (625,260)-(656,291): text "62"; invisible if not DALI_Config.Kurzadr[62]; alarm colour if DALI_Config.LampeEin[62]
rectangle at (465,260)-(496,291): text "58"; alarm colour if DALI_Config.Kurzadr[58]
rectangle at (465,260)-(496,291): text "58"; invisible if not DALI_Config.Kurzadr[58]; alarm colour if DALI_Config.LampeEin[58]
rectangle at (665,260)-(696,291): text "63"; alarm colour if DALI_Config.Kurzadr[63]
rectangle at (665,260)-(696,291): text "63"; invisible if not DALI_Config.Kurzadr[63]; alarm colour if DALI_Config.LampeEin[63]
rectangle at (705,260)-(736,291): text "64"; alarm colour if DALI_Config.Kurzadr[64]
rectangle at (705,260)-(736,291): text "64"; invisible if not DALI_Config.Kurzadr[64]; alarm colour if DALI_Config.LampeEin[64]
rectangle at (80,310)-(761,496): text "Lamp failure"
rectangle at (105,335)-(136,366): text "1"; alarm colour if DALI_Config.Kurzadr[1]
rectangle at (105,335)-(136,366): text "1"; invisible if not DALI_Config.Kurzadr[1]; alarm colour if DALI_Config.Lampenausfall[1]
rectangle at (145,335)-(176,366): text "2"; alarm colour if DALI_Config.Kurzadr[2]
rectangle at (145,335)-(176,366): text "2"; invisible if not DALI_Config.Kurzadr[2]; alarm colour if DALI_Config.Lampenausfall[2]
rectangle at (185,335)-(216,366): text "3"; alarm colour if DALI_Config.Kurzadr[3]
rectangle at (185,335)-(216,366): text "3"; invisible if not DALI_Config.Kurzadr[3]; alarm colour if DALI_Config.Lampenausfall[3]
rectangle at (225,335)-(256,366): text "4"; alarm colour if DALI_Config.Kurzadr[4]
rectangle at (225,335)-(256,366): text "4"; invisible if not DALI_Config.Kurzadr[4]; alarm colour if DALI_Config.Lampenausfall[4]
rectangle at (265,335)-(296,366): text "5"; alarm colour if DALI_Config.Kurzadr[5]
rectangle at (265,335)-(296,366): text "5"; invisible if not DALI_Config.Kurzadr[5]; alarm colour if DALI_Config.Lampenausfall[5]
rectangle at (305,335)-(336,366): text "6"; alarm colour if DALI_Config.Kurzadr[6]
rectangle at (305,335)-(336,366): text "6"; invisible if not DALI_Config.Kurzadr[6]; alarm colour if DALI_Config.Lampenausfall[6]
rectangle at (345,335)-(376,366): text "7"; alarm colour if DALI_Config.Kurzadr[7]
rectangle at (345,335)-(376,366): text "7"; invisible if not DALI_Config.Kurzadr[7]; alarm colour if DALI_Config.Lampenausfall[7]
rectangle at (385,335)-(416,366): text "8"; alarm colour if DALI_Config.Kurzadr[8]
rectangle at (385,335)-(416,366): text "8"; invisible if not DALI_Config.Kurzadr[8]; alarm colour if DALI_Config.Lampenausfall[8]
rectangle at (425,335)-(456,366): text "9"; alarm colour if DALI_Config.Kurzadr[9]
rectangle at (425,335)-(456,366): text "9"; invisible if not DALI_Config.Kurzadr[9]; alarm colour if DALI_Config.Lampenausfall[9]
rectangle at (465,335)-(496,366): text "10"; alarm colour if DALI_Config.Kurzadr[10]
rectangle at (465,335)-(496,366): text "10"; invisible if not DALI_Config.Kurzadr[10]; alarm colour if DALI_Config.Lampenausfall[10]
rectangle at (505,335)-(536,366): text "11"; alarm colour if DALI_Config.Kurzadr[11]
rectangle at (505,335)-(536,366): text "11"; invisible if not DALI_Config.Kurzadr[11]; alarm colour if DALI_Config.Lampenausfall[11]
rectangle at (545,335)-(576,366): text "12"; alarm colour if DALI_Config.Kurzadr[12]
rectangle at (545,335)-(576,366): text "12"; invisible if not DALI_Config.Kurzadr[12]; alarm colour if DALI_Config.Lampenausfall[12]
rectangle at (585,335)-(616,366): text "13"; alarm colour if DALI_Config.Kurzadr[13]
rectangle at (585,335)-(616,366): text "13"; invisible if not DALI_Config.Kurzadr[13]; alarm colour if DALI_Config.Lampenausfall[13]
rectangle at (625,335)-(656,366): text "14"; alarm colour if DALI_Config.Kurzadr[14]
rectangle at (625,335)-(656,366): text "14"; invisible if not DALI_Config.Kurzadr[14]; alarm colour if DALI_Config.Lampenausfall[14]
rectangle at (665,335)-(696,366): text "15"; alarm colour if DALI_Config.Kurzadr[15]
rectangle at (665,335)-(696,366): text "15"; invisible if not DALI_Config.Kurzadr[15]; alarm colour if DALI_Config.Lampenausfall[15]
rectangle at (705,335)-(736,366): text "16"; alarm colour if DALI_Config.Kurzadr[16]
rectangle at (705,335)-(736,366): text "16"; invisible if not DALI_Config.Kurzadr[16]; alarm colour if DALI_Config.Lampenausfall[16]
rectangle at (105,375)-(136,406): text "17"; alarm colour if DALI_Config.Kurzadr[17]
rectangle at (105,375)-(136,406): text "17"; invisible if not DALI_Config.Kurzadr[17]; alarm colour if DALI_Config.Lampenausfall[17]
rectangle at (185,375)-(216,406): text "19"; alarm colour if DALI_Config.Kurzadr[19]
rectangle at (185,375)-(216,406): text "19"; invisible if not DALI_Config.Kurzadr[19]; alarm colour if DALI_Config.Lampenausfall[19]
rectangle at (145,375)-(176,406): text "18"; alarm colour if DALI_Config.Kurzadr[18]
rectangle at (145,375)-(176,406): text "18"; invisible if not DALI_Config.Kurzadr[18]; alarm colour if DALI_Config.Lampenausfall[18]
rectangle at (225,375)-(256,406): text "20"; alarm colour if DALI_Config.Kurzadr[20]
rectangle at (225,375)-(256,406): text "20"; invisible if not DALI_Config.Kurzadr[20]; alarm colour if DALI_Config.Lampenausfall[20]
rectangle at (265,375)-(296,406): text "21"; alarm colour if DALI_Config.Kurzadr[21]
rectangle at (265,375)-(296,406): text "21"; invisible if not DALI_Config.Kurzadr[21]; alarm colour if DALI_Config.Lampenausfall[21]
rectangle at (305,375)-(336,406): text "22"; alarm colour if DALI_Config.Kurzadr[22]
rectangle at (305,375)-(336,406): text "22"; invisible if not DALI_Config.Kurzadr[22]; alarm colour if DALI_Config.Lampenausfall[22]
rectangle at (345,375)-(376,406): text "23"; alarm colour if DALI_Config.Kurzadr[23]
rectangle at (345,375)-(376,406): text "23"; invisible if not DALI_Config.Kurzadr[23]; alarm colour if DALI_Config.Lampenausfall[23]
rectangle at (385,375)-(416,406): text "24"; alarm colour if DALI_Config.Kurzadr[24]
rectangle at (385,375)-(416,406): text "24"; invisible if not DALI_Config.Kurzadr[24]; alarm colour if DALI_Config.Lampenausfall[24]
rectangle at (425,375)-(456,406): text "25"; alarm colour if DALI_Config.Kurzadr[25]
rectangle at (425,375)-(456,406): text "25"; invisible if not DALI_Config.Kurzadr[25]; alarm colour if DALI_Config.Lampenausfall[25]
rectangle at (585,375)-(616,406): text "29"; alarm colour if DALI_Config.Kurzadr[29]
rectangle at (585,375)-(616,406): text "29"; invisible if not DALI_Config.Kurzadr[29]; alarm colour if DALI_Config.Lampenausfall[29]
rectangle at (545,375)-(576,406): text "28"; alarm colour if DALI_Config.Kurzadr[28]
rectangle at (545,375)-(576,406): text "28"; invisible if not DALI_Config.Kurzadr[28]; alarm colour if DALI_Config.Lampenausfall[28]
rectangle at (505,375)-(536,406): text "27"; alarm colour if DALI_Config.Kurzadr[27]
rectangle at (505,375)-(536,406): text "27"; invisible if not DALI_Config.Kurzadr[27]; alarm colour if DALI_Config.Lampenausfall[27]
rectangle at (465,375)-(496,406): text "26"; alarm colour if DALI_Config.Kurzadr[26]
rectangle at (465,375)-(496,406): text "26"; invisible if not DALI_Config.Kurzadr[26]; alarm colour if DALI_Config.Lampenausfall[26]
rectangle at (625,375)-(656,406): text "30"; alarm colour if DALI_Config.Kurzadr[30]
rectangle at (625,375)-(656,406): text "30"; invisible if not DALI_Config.Kurzadr[30]; alarm colour if DALI_Config.Lampenausfall[30]
rectangle at (665,375)-(696,406): text "31"; alarm colour if DALI_Config.Kurzadr[31]
rectangle at (665,375)-(696,406): text "31"; invisible if not DALI_Config.Kurzadr[31]; alarm colour if DALI_Config.Lampenausfall[31]
rectangle at (705,375)-(736,406): text "32"; alarm colour if DALI_Config.Kurzadr[32]
rectangle at (705,375)-(736,406): text "32"; invisible if not DALI_Config.Kurzadr[32]; alarm colour if DALI_Config.Lampenausfall[32]
rectangle at (105,415)-(136,446): text "33"; alarm colour if DALI_Config.Kurzadr[33]
rectangle at (105,415)-(136,446): text "33"; invisible if not DALI_Config.Kurzadr[33]; alarm colour if DALI_Config.Lampenausfall[33]
rectangle at (145,415)-(176,446): text "34"; alarm colour if DALI_Config.Kurzadr[34]
rectangle at (145,415)-(176,446): text "34"; invisible if not DALI_Config.Kurzadr[34]; alarm colour if DALI_Config.Lampenausfall[34]
rectangle at (225,415)-(256,446): text "36"; alarm colour if DALI_Config.Kurzadr[36]
rectangle at (225,415)-(256,446): text "36"; invisible if not DALI_Config.Kurzadr[36]; alarm colour if DALI_Config.Lampenausfall[36]
rectangle at (305,415)-(336,446): text "38"; alarm colour if DALI_Config.Kurzadr[38]
rectangle at (305,415)-(336,446): text "38"; invisible if not DALI_Config.Kurzadr[38]; alarm colour if DALI_Config.Lampenausfall[38]
rectangle at (345,415)-(376,446): text "39"; alarm colour if DALI_Config.Kurzadr[39]
rectangle at (345,415)-(376,446): text "39"; invisible if not DALI_Config.Kurzadr[39]; alarm colour if DALI_Config.Lampenausfall[39]
rectangle at (265,415)-(296,446): text "37"; alarm colour if DALI_Config.Kurzadr[37]
rectangle at (265,415)-(296,446): text "37"; invisible if not DALI_Config.Kurzadr[37]; alarm colour if DALI_Config.Lampenausfall[37]
rectangle at (185,415)-(216,446): text "35"; alarm colour if DALI_Config.Kurzadr[35]
rectangle at (185,415)-(216,446): text "35"; invisible if not DALI_Config.Kurzadr[35]; alarm colour if DALI_Config.Lampenausfall[35]
rectangle at (425,415)-(456,446): text "41"; alarm colour if DALI_Config.Kurzadr[41]
rectangle at (425,415)-(456,446): text "41"; invisible if not DALI_Config.Kurzadr[41]; alarm colour if DALI_Config.Lampenausfall[41]
rectangle at (465,415)-(496,446): text "42"; alarm colour if DALI_Config.Kurzadr[42]
rectangle at (465,415)-(496,446): text "42"; invisible if not DALI_Config.Kurzadr[42]; alarm colour if DALI_Config.Lampenausfall[42]
rectangle at (385,415)-(416,446): text "40"; alarm colour if DALI_Config.Kurzadr[40]
rectangle at (385,415)-(416,446): text "40"; invisible if not DALI_Config.Kurzadr[40]; alarm colour if DALI_Config.Lampenausfall[40]
rectangle at (505,415)-(536,446): text "43"; alarm colour if DALI_Config.Kurzadr[43]
rectangle at (505,415)-(536,446): text "43"; invisible if not DALI_Config.Kurzadr[43]; alarm colour if DALI_Config.Lampenausfall[43]
rectangle at (545,415)-(576,446): text "44"; alarm colour if DALI_Config.Kurzadr[44]
rectangle at (545,415)-(576,446): text "44"; invisible if not DALI_Config.Kurzadr[44]; alarm colour if DALI_Config.Lampenausfall[44]
rectangle at (585,415)-(616,446): text "45"; alarm colour if DALI_Config.Kurzadr[45]
rectangle at (585,415)-(616,446): text "45"; invisible if not DALI_Config.Kurzadr[45]; alarm colour if DALI_Config.Lampenausfall[45]
rectangle at (625,415)-(656,446): text "46"; alarm colour if DALI_Config.Kurzadr[46]
rectangle at (625,415)-(656,446): text "46"; invisible if not DALI_Config.Kurzadr[46]; alarm colour if DALI_Config.Lampenausfall[46]
rectangle at (665,415)-(696,446): text "47"; alarm colour if DALI_Config.Kurzadr[47]
rectangle at (665,415)-(696,446): text "47"; invisible if not DALI_Config.Kurzadr[47]; alarm colour if DALI_Config.Lampenausfall[47]
rectangle at (705,415)-(736,446): text "48"; alarm colour if DALI_Config.Kurzadr[48]
rectangle at (705,415)-(736,446): text "48"; invisible if not DALI_Config.Kurzadr[48]; alarm colour if DALI_Config.Lampenausfall[48]
rectangle at (105,455)-(136,486): text "49"; alarm colour if DALI_Config.Kurzadr[49]
rectangle at (105,455)-(136,486): text "49"; invisible if not DALI_Config.Kurzadr[49]; alarm colour if DALI_Config.Lampenausfall[49]
rectangle at (145,455)-(176,486): text "50"; alarm colour if DALI_Config.Kurzadr[50]
rectangle at (145,455)-(176,486): text "50"; invisible if not DALI_Config.Kurzadr[50]; alarm colour if DALI_Config.Lampenausfall[50]
rectangle at (185,455)-(216,486): text "51"; alarm colour if DALI_Config.Kurzadr[51]
rectangle at (185,455)-(216,486): text "51"; invisible if not DALI_Config.Kurzadr[51]; alarm colour if DALI_Config.Lampenausfall[51]
rectangle at (225,455)-(256,486): text "52"; alarm colour if DALI_Config.Kurzadr[52]
rectangle at (225,455)-(256,486): text "52"; invisible if not DALI_Config.Kurzadr[52]; alarm colour if DALI_Config.Lampenausfall[52]
rectangle at (265,455)-(296,486): text "53"; alarm colour if DALI_Config.Kurzadr[53]
rectangle at (265,455)-(296,486): text "53"; invisible if not DALI_Config.Kurzadr[53]; alarm colour if DALI_Config.Lampenausfall[53]
rectangle at (305,455)-(336,486): text "54"; alarm colour if DALI_Config.Kurzadr[54]
rectangle at (305,455)-(336,486): text "54"; invisible if not DALI_Config.Kurzadr[54]; alarm colour if DALI_Config.Lampenausfall[54]
rectangle at (345,455)-(376,486): text "55"; alarm colour if DALI_Config.Kurzadr[55]
rectangle at (345,455)-(376,486): text "55"; invisible if not DALI_Config.Kurzadr[55]; alarm colour if DALI_Config.Lampenausfall[55]
rectangle at (385,455)-(416,486): text "56"; alarm colour if DALI_Config.Kurzadr[56]
rectangle at (385,455)-(416,486): text "56"; invisible if not DALI_Config.Kurzadr[56]; alarm colour if DALI_Config.Lampenausfall[56]
rectangle at (425,455)-(456,486): text "57"; alarm colour if DALI_Config.Kurzadr[57]
rectangle at (425,455)-(456,486): text "57"; invisible if not DALI_Config.Kurzadr[57]; alarm colour if DALI_Config.Lampenausfall[57]
rectangle at (505,455)-(536,486): text "59"; alarm colour if DALI_Config.Kurzadr[59]
rectangle at (505,455)-(536,486): text "59"; invisible if not DALI_Config.Kurzadr[59]; alarm colour if DALI_Config.Lampenausfall[59]
rectangle at (545,455)-(576,486): text "60"; alarm colour if DALI_Config.Kurzadr[60]
rectangle at (545,455)-(576,486): text "60"; invisible if not DALI_Config.Kurzadr[60]; alarm colour if DALI_Config.Lampenausfall[60]
rectangle at (585,455)-(616,486): text "61"; alarm colour if DALI_Config.Kurzadr[61]
rectangle at (585,455)-(616,486): text "61"; invisible if not DALI_Config.Kurzadr[61]; alarm colour if DALI_Config.Lampenausfall[61]
rectangle at (625,455)-(656,486): text "62"; alarm colour if DALI_Config.Kurzadr[62]
rectangle at (625,455)-(656,486): text "62"; invisible if not DALI_Config.Kurzadr[62]; alarm colour if DALI_Config.Lampenausfall[62]
rectangle at (465,455)-(496,486): text "58"; alarm colour if DALI_Config.Kurzadr[58]
rectangle at (465,455)-(496,486): text "58"; invisible if not DALI_Config.Kurzadr[58]; alarm colour if DALI_Config.Lampenausfall[58]
rectangle at (665,455)-(696,486): text "63"; alarm colour if DALI_Config.Kurzadr[63]
rectangle at (665,455)-(696,486): text "63"; invisible if not DALI_Config.Kurzadr[63]; alarm colour if DALI_Config.Lampenausfall[63]
rectangle at (705,455)-(736,486): text "64"; alarm colour if DALI_Config.Kurzadr[64]
rectangle at (705,455)-(736,486): text "64"; invisible if not DALI_Config.Kurzadr[64]; alarm colour if DALI_Config.Lampenausfall[64]
button at (345,505)-(496,541): text "Query status"; taps DALI_Config.Status; tooltip If you click the button "Query Status", you will get the status "Lamp failure" and "Lamp arc power on" from the ECG.
rectangle at (110,505)-(271,526): text "Short address available"
rectangle at (125,535)-(256,556): text "Lamp failure"
rectangle at (125,565)-(196,586): text "Lamp on"
6 more shapes without text or variables
*)

(* Visualisation lux
rectangle at (915,525)-(1011,546): text "Zpet"; opens PLC_VISU; tooltip Back to home page
1 elements of other kinds (tables, trends, ...) not read
*)

(* Visualisation PLC_VISU
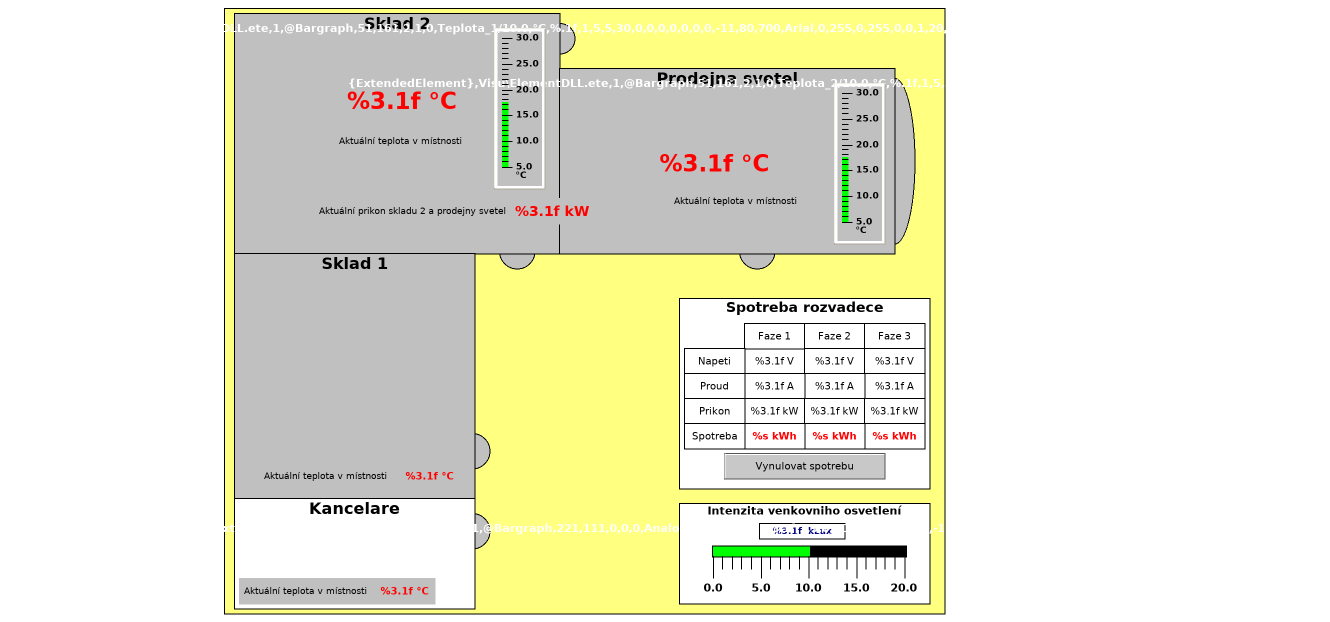
ellipse at (545,225)-(581,261): alarm colour if .KA13; taps .TL10s; tooltip Dlouhý stisk zapne svìtlo. (cca 1s)
ellipse at (305,225)-(341,261): alarm colour if .KA16; taps .TL05s; tooltip Dlouhý stisk zapne svìtlo. (cca 1s)
ellipse at (350,15)-(381,46): alarm colour if .KA15; taps .TL06s; tooltip Dlouhý stisk zapne svìtlo. (cca 1s)
rectangle at (40,5)-(366,246): text "Sklad 2"; opens DALI_cfg
rectangle at (40,245)-(281,491): text "Sklad 1"; opens DALI_cfg
rectangle at (365,60)-(701,246): text "Prodejna svetel"; opens prodej_svetel
rectangle at (40,490)-(281,601): text "Kancelare"
rectangle at (65,455)-(206,481): text "Aktuální teplota v místnosti"
rectangle at (205,455)-(266,481): text "%3.1f °C"; shows .Teplota_3/10.0
rectangle at (140,120)-(281,146): text "Aktuální teplota v místnosti"
rectangle at (150,65)-(266,121): text "%3.1f °C"; shows .Teplota_1/10.0
rectangle at (465,125)-(576,186): text "%3.1f °C"; shows .Teplota_2/10.0
rectangle at (475,180)-(611,206): text "Aktuální teplota v místnosti"
rectangle at (45,570)-(181,596): text "Aktuální teplota v místnosti"
rectangle at (180,570)-(241,596): text "%3.1f °C"; shows .Teplota_4/10.0
rounded rectangle at (485,290)-(736,481): text "Spotreba rozvadece"
rectangle at (550,340)-(611,366): text "%3.1f V"; shows TriFaze.arNapeti[1]
rectangle at (550,315)-(611,341): text "Faze 1"
rectangle at (610,315)-(671,341): text "Faze 2"
rectangle at (670,315)-(731,341): text "Faze 3"
rectangle at (610,340)-(671,366): text "%3.1f V"; shows TriFaze.arNapeti[2]
rectangle at (670,340)-(731,366): text "%3.1f V"; shows TriFaze.arNapeti[3]
rectangle at (670,365)-(731,391): text "%3.1f A"; shows TriFaze.arProud[3]
rectangle at (610,365)-(671,391): text "%3.1f A"; shows TriFaze.arProud[2]
rectangle at (550,365)-(611,391): text "%3.1f A"; shows TriFaze.arProud[1]
rectangle at (550,390)-(611,416): text "%3.1f kW"; shows TriFaze.arVykon[1]
rectangle at (610,390)-(671,416): text "%3.1f kW"; shows TriFaze.arVykon[2]
rectangle at (670,390)-(731,416): text "%3.1f kW"; shows TriFaze.arVykon[3]
rectangle at (670,415)-(731,441): text "%s kWh"; shows TriFaze.adwSpotreba[3]
rectangle at (610,415)-(671,441): text "%s kWh"; shows TriFaze.adwSpotreba[2]
rectangle at (550,415)-(611,441): text "%s kWh"; shows TriFaze.adwSpotreba[1]
button at (530,445)-(691,471): text "Vynulovat spotrebu"; taps TriFaze.SmazL1
rounded rectangle at (485,495)-(736,596): text "Intenzita venkovniho osvetlení"; opens lux
rectangle at (565,515)-(651,531): text "%3.1f  kLux"; shows .Analog_1/3276.4*2
rectangle at (490,340)-(551,366): text "Napeti"
rectangle at (490,365)-(551,391): text "Proud"
rectangle at (490,390)-(551,416): text "Prikon"
rectangle at (490,415)-(551,441): text "Spotreba"
rectangle at (120,190)-(331,216): text "Aktuální prikon skladu 2 a prodejny svetel"
rectangle at (325,190)-(391,216): text "%3.1f kW"; shows TriFaze.arVykon[1]+TriFaze.arVykon[2]+TriFaze.arVykon[3]
group at (505,520)-(726,621)
  rectangle at (0,0)-(1,1): text "{ExtendedElement},Visu\ElementDLL.ete,1,@Bargraph,221,111,0,0,0,Analog_1/3276.4*2,,%.1f,1,5,0,20,0,0,0,0,0,0,0,-13,16,700,Arial,0,255,0,255,0,0,0,0,1,0,0,"
  rectangle at (14,19)-(111,29): alarm colour if (Analog_1/3276.4*2) < 0; right ((Analog_1/3276.4*2 * 1.0) - 10)  * 9.6
  rectangle at (2,53)-(26,103): text "0.0"
  rectangle at (50,53)-(74,103): text "5.0"
  rectangle at (93,53)-(126,103): text "10.0"
  rectangle at (141,53)-(174,103): text "15.0"
  rectangle at (189,53)-(222,103): text "20.0"
group at (640,75)-(691,236)
  rectangle at (0,0)-(1,1): text "{ExtendedElement},Visu\ElementDLL.ete,1,@Bargraph,51,161,2,1,0,Teplota_2/10.0,°C,%.1f,1,5,5,30,0,0,0,0,0,0,0,-11,80,700,Arial,0,255,0,255,0,0,1,25,0,1,0,"
  rectangle at (8,74)-(14,139): alarm colour if (Teplota_2/10.0) > 25; top ((Teplota_2/10.0 * 1.0) - 17.5)  * -5.2
  rectangle at (20,129)-(47,148): text "5.0"
  rectangle at (20,103)-(47,122): text "10.0"
  rectangle at (20,77)-(47,96): text "15.0"
  rectangle at (20,52)-(47,71): text "20.0"
  rectangle at (20,26)-(47,45): text "25.0"
  rectangle at (20,0)-(47,19): text "30.0"
  rectangle at (15,140)-(39,154): text "°C"
group at (300,20)-(351,181)
  rectangle at (0,0)-(1,1): text "{ExtendedElement},Visu\ElementDLL.ete,1,@Bargraph,51,161,2,1,0,Teplota_1/10.0,°C,%.1f,1,5,5,30,0,0,0,0,0,0,0,-11,80,700,Arial,0,255,0,255,0,0,1,20,0,1,0,"
  rectangle at (8,74)-(14,139): alarm colour if (Teplota_1/10.0) > 20; top ((Teplota_1/10.0 * 1.0) - 17.5)  * -5.2
  rectangle at (20,129)-(47,148): text "5.0"
  rectangle at (20,103)-(47,122): text "10.0"
  rectangle at (20,77)-(47,96): text "15.0"
  rectangle at (20,52)-(47,71): text "20.0"
  rectangle at (20,26)-(47,45): text "25.0"
  rectangle at (20,0)-(47,19): text "30.0"
  rectangle at (15,140)-(39,154): text "°C"
94 more shapes without text or variables
*)

(* Visualisation prodej_svetel
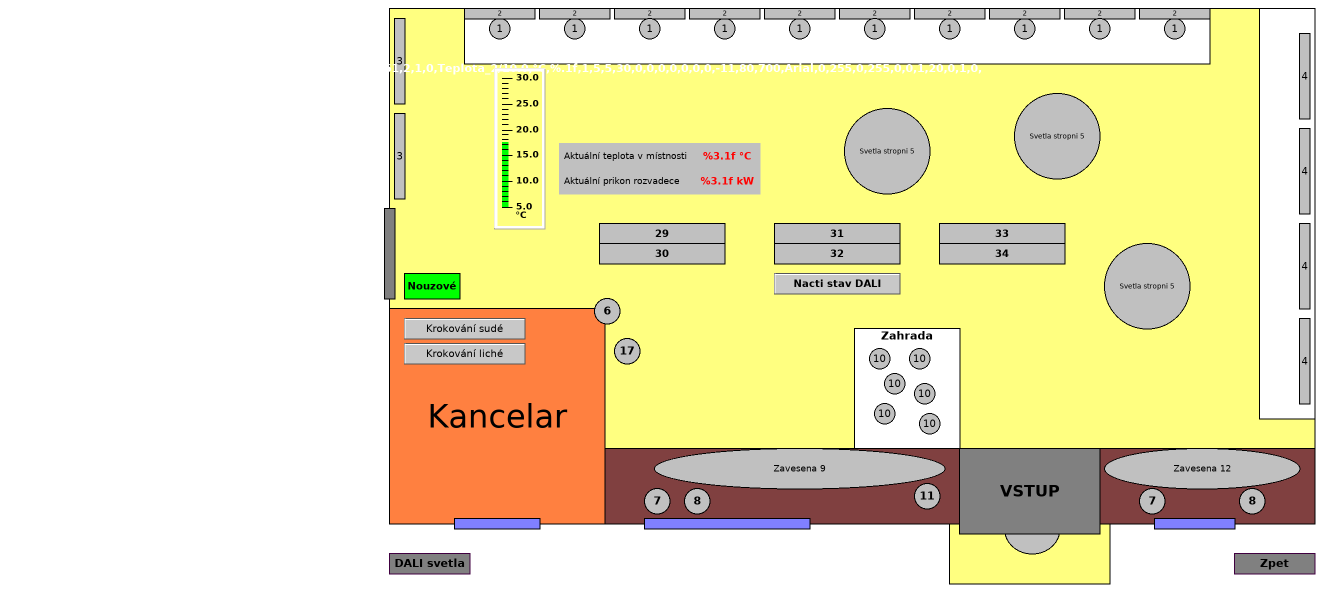
rounded rectangle at (485,345)-(591,476): text "Zahrada"
ellipse at (635,520)-(691,571): alarm colour if .KA13; taps .TL10s; tooltip Dlouhý stisk zapne svìtlo. (cca 1s)
rectangle at (25,130)-(36,216): text "3"; alarm colour if .KA03
rectangle at (35,290)-(91,316): text "Nouzové"; alarm colour if .KA20
rectangle at (20,325)-(236,541): text "Kancelar"
rectangle at (865,570)-(946,591): text "Zpet"; opens PLC_VISU; tooltip Back to home page
ellipse at (315,505)-(341,531): text "8"; alarm colour if .ka08
ellipse at (735,465)-(931,506): text "Zavesena 12"; alarm colour if .KA12
rectangle at (930,50)-(941,136): text "4"; alarm colour if .KA04
ellipse at (500,365)-(521,386): text "10"; alarm colour if .KA10
ellipse at (285,465)-(576,506): text "Zavesena 9"; alarm colour if .KA09
rectangle at (590,465)-(731,551): text "VSTUP"
rectangle at (325,160)-(391,186): text "%3.1f °C"; shows .Teplota_2/10.0
rectangle at (190,160)-(326,186): text "Aktuální teplota v místnosti"
ellipse at (120,35)-(141,56): text "1"; alarm colour if .KA01; taps .TL10s; tooltip Klinutím zapínáte žárovky na deskách
rectangle at (95,25)-(166,36): text "2"; alarm colour if .KA02
ellipse at (275,505)-(301,531): text "7"; alarm colour if .ka07
ellipse at (870,505)-(896,531): text "8"; alarm colour if .ka08
ellipse at (770,505)-(796,531): text "7"; alarm colour if .ka07
rectangle at (930,145)-(941,231): text "4"; alarm colour if .KA04
rectangle at (930,335)-(941,421): text "4"; alarm colour if .KA04
rectangle at (930,240)-(941,326): text "4"; alarm colour if .KA04
rectangle at (25,35)-(36,121): text "3"; alarm colour if .KA03
rectangle at (190,185)-(326,211): text "Aktuální prikon rozvadece"
rectangle at (325,185)-(391,211): text "%3.1f kW"; shows TriFaze.arVykon[1]+TriFaze.arVykon[2]+TriFaze.arVykon[3]
button at (35,335)-(156,356): text "Krokování sudé"; taps .TL08s; tooltip Kliknutím krokujete sudé releové výstupy oovládající svìtla.
button at (35,360)-(156,381): text "Krokování liché"; taps .TL07s; tooltip Kliknutím krokujete liché releové výstupy oovládající svìtla.
rectangle at (230,240)-(356,261): text "29"; alarm colour if DALI_Config.Kurzadr[29]
rectangle at (230,240)-(356,261): text "29"; invisible if not DALI_Config.Kurzadr[29]; alarm colour if DALI_Config.LampeEin[29]; taps .TL09s; tooltip Kliknutím zapínáte a vypínáte svìtla DALI
rectangle at (230,260)-(356,281): text "30"; alarm colour if DALI_Config.Kurzadr[30]
rectangle at (230,260)-(356,281): text "30"; invisible if not DALI_Config.Kurzadr[30]; alarm colour if DALI_Config.LampeEin[30]; taps .TL09s; tooltip Kliknutím zapínáte a vypínáte svìtla DALI
rectangle at (405,240)-(531,261): text "31"; alarm colour if DALI_Config.Kurzadr[31]
rectangle at (405,240)-(531,261): text "31"; invisible if not DALI_Config.Kurzadr[31]; alarm colour if DALI_Config.LampeEin[31]; taps .TL09s; tooltip Kliknutím zapínáte a vypínáte svìtla DALI
rectangle at (405,260)-(531,281): text "32"; alarm colour if DALI_Config.Kurzadr[32]
rectangle at (405,260)-(531,281): text "32"; invisible if not DALI_Config.Kurzadr[32]; alarm colour if DALI_Config.LampeEin[32]; taps .TL09s; tooltip Kliknutím zapínáte a vypínáte svìtla DALI
rectangle at (570,240)-(696,261): text "33"; alarm colour if DALI_Config.Kurzadr[33]
rectangle at (570,240)-(696,261): text "33"; invisible if not DALI_Config.Kurzadr[33]; alarm colour if DALI_Config.LampeEin[33]; taps .TL09s; tooltip Kliknutím zapínáte a vypínáte svìtla DALI
rectangle at (570,260)-(696,281): text "34"; alarm colour if DALI_Config.Kurzadr[34]
rectangle at (570,260)-(696,281): text "34"; invisible if not DALI_Config.Kurzadr[34]; alarm colour if DALI_Config.LampeEin[34]; taps .TL09s; tooltip Kliknutím zapínáte a vypínáte svìtla DALI
button at (405,290)-(531,311): text "Nacti stav DALI"; taps DALI_Config.Status; tooltip Kliknutim nactete status svetel. (sviti, nesviti, vadna).
rectangle at (245,25)-(316,36): text "2"; alarm colour if .KA02
ellipse at (195,35)-(216,56): text "1"; alarm colour if .KA01; taps .TL10s; tooltip Klinutím zapínáte žárovky na deskách
rectangle at (170,25)-(241,36): text "2"; alarm colour if .KA02
ellipse at (270,35)-(291,56): text "1"; alarm colour if .KA01; taps .TL10s; tooltip Klinutím zapínáte žárovky na deskách
ellipse at (345,35)-(366,56): text "1"; alarm colour if .KA01; taps .TL10s; tooltip Klinutím zapínáte žárovky na deskách
rectangle at (320,25)-(391,36): text "2"; alarm colour if .KA02
rectangle at (470,25)-(541,36): text "2"; alarm colour if .KA02
ellipse at (420,35)-(441,56): text "1"; alarm colour if .KA01; taps .TL10s; tooltip Klinutím zapínáte žárovky na deskách
rectangle at (395,25)-(466,36): text "2"; alarm colour if .KA02
ellipse at (495,35)-(516,56): text "1"; alarm colour if .KA01; taps .TL10s; tooltip Klinutím zapínáte žárovky na deskách
ellipse at (570,35)-(591,56): text "1"; alarm colour if .KA01; taps .TL10s; tooltip Klinutím zapínáte žárovky na deskách
rectangle at (545,25)-(616,36): text "2"; alarm colour if .KA02
rectangle at (695,25)-(766,36): text "2"; alarm colour if .KA02
ellipse at (645,35)-(666,56): text "1"; alarm colour if .KA01; taps .TL10s; tooltip Klinutím zapínáte žárovky na deskách
rectangle at (620,25)-(691,36): text "2"; alarm colour if .KA02
ellipse at (720,35)-(741,56): text "1"; alarm colour if .KA01; taps .TL10s; tooltip Klinutím zapínáte žárovky na deskách
ellipse at (795,35)-(816,56): text "1"; alarm colour if .KA01; taps .TL10s; tooltip Klinutím zapínáte žárovky na deskách
rectangle at (770,25)-(841,36): text "2"; alarm colour if .KA02
ellipse at (475,125)-(561,211): text "Svetla stropni 5"; alarm colour if .KA05
ellipse at (645,110)-(731,196): text "Svetla stropni 5"; alarm colour if .KA05
ellipse at (735,260)-(821,346): text "Svetla stropni 5"; alarm colour if .KA05
ellipse at (505,420)-(526,441): text "10"; alarm colour if .KA10
ellipse at (545,400)-(566,421): text "10"; alarm colour if .KA10
ellipse at (540,365)-(561,386): text "10"; alarm colour if .KA10
ellipse at (550,430)-(571,451): text "10"; alarm colour if .KA10
ellipse at (515,390)-(536,411): text "10"; alarm colour if .KA10
ellipse at (225,315)-(251,341): text "6"; alarm colour if .ka06
ellipse at (545,500)-(571,526): text "11"; alarm colour if .ka11
ellipse at (245,355)-(271,381): text "17"; alarm colour if .ka17
group at (125,85)-(176,246)
  rectangle at (0,0)-(1,1): text "{ExtendedElement},Visu\ElementDLL.ete,1,@Bargraph,51,161,2,1,0,Teplota_2/10.0,°C,%.1f,1,5,5,30,0,0,0,0,0,0,0,-11,80,700,Arial,0,255,0,255,0,0,1,20,0,1,0,"
  rectangle at (8,74)-(14,139): alarm colour if (Teplota_2/10.0) > 20; top ((Teplota_2/10.0 * 1.0) - 17.5)  * -5.2
  rectangle at (20,129)-(47,148): text "5.0"
  rectangle at (20,103)-(47,122): text "10.0"
  rectangle at (20,77)-(47,96): text "15.0"
  rectangle at (20,52)-(47,71): text "20.0"
  rectangle at (20,26)-(47,45): text "25.0"
  rectangle at (20,0)-(47,19): text "30.0"
  rectangle at (15,140)-(39,154): text "°C"
rectangle at (20,570)-(101,591): text "DALI svetla"; opens DALI_cfg; tooltip Back to home page
44 more shapes without text or variables
*)

(* Visualisation Scene_configuration
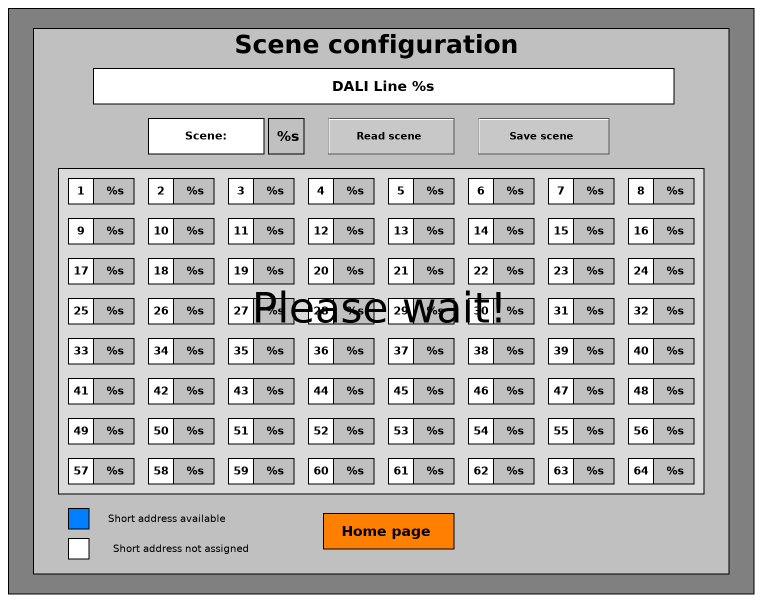
rectangle at (50,25)-(746,571): text "Scene configuration"
rounded rectangle at (340,510)-(471,546): text "Home page"; opens DALI; tooltip Back to home page
rounded rectangle at (110,65)-(691,101): text "DALI Line %s"; shows DALI_Config.bDali_Linie; tooltip You can change the DALI Line only on the home page.
rectangle at (85,175)-(111,201): text "1"; alarm colour if Dali_Config.Kurzadr[1]
rectangle at (110,175)-(151,201): text "%s"; shows DALI_Config.Szenenwert[1]; tooltip 0 % = Off 1 - 100 % = Dim level 101 % = Mask; editable
button at (495,115)-(626,151): text "Save scene"; taps DALI_Config.SzeneSpeichern; tooltip Save the configured dim levels in the ECGs.
button at (345,115)-(471,151): text "Read scene"; taps DALI_Config.SzeneLesen; tooltip Read the saved scene values from the ECGs.
rectangle at (85,215)-(111,241): text "9"; alarm colour if Dali_Config.Kurzadr[9]
rectangle at (110,215)-(151,241): text "%s"; shows DALI_Config.Szenenwert[9]; tooltip 0 % = Off 1 - 100 % = Dim level 101 % = Mask; editable
rectangle at (85,255)-(111,281): text "17"; alarm colour if Dali_Config.Kurzadr[17]
rectangle at (110,255)-(151,281): text "%s"; shows DALI_Config.Szenenwert[17]; tooltip 0 % = Off 1 - 100 % = Dim level 101 % = Mask; editable
rectangle at (85,295)-(111,321): text "25"; alarm colour if Dali_Config.Kurzadr[25]
rectangle at (110,295)-(151,321): text "%s"; shows DALI_Config.Szenenwert[25]; tooltip 0 % = Off 1 - 100 % = Dim level 101 % = Mask; editable
rectangle at (85,335)-(111,361): text "33"; alarm colour if Dali_Config.Kurzadr[33]
rectangle at (110,335)-(151,361): text "%s"; shows DALI_Config.Szenenwert[33]; tooltip 0 % = Off 1 - 100 % = Dim level 101 % = Mask; editable
rectangle at (85,375)-(111,401): text "41"; alarm colour if Dali_Config.Kurzadr[41]
rectangle at (110,375)-(151,401): text "%s"; shows DALI_Config.Szenenwert[41]; tooltip 0 % = Off 1 - 100 % = Dim level 101 % = Mask; editable
rectangle at (85,415)-(111,441): text "49"; alarm colour if Dali_Config.Kurzadr[49]
rectangle at (110,415)-(151,441): text "%s"; shows DALI_Config.Szenenwert[49]; tooltip 0 % = Off 1 - 100 % = Dim level 101 % = Mask; editable
rectangle at (85,455)-(111,481): text "57"; alarm colour if Dali_Config.Kurzadr[57]
rectangle at (110,455)-(151,481): text "%s"; shows DALI_Config.Szenenwert[57]; tooltip 0 % = Off 1 - 100 % = Dim level 101 % = Mask; editable
rectangle at (165,175)-(191,201): text "2"; alarm colour if Dali_Config.Kurzadr[2]
rectangle at (190,175)-(231,201): text "%s"; shows DALI_Config.Szenenwert[2]; tooltip 0 % = Off 1 - 100 % = Dim level 101 % = Mask; editable
rectangle at (165,215)-(191,241): text "10"; alarm colour if Dali_Config.Kurzadr[10]
rectangle at (190,215)-(231,241): text "%s"; shows DALI_Config.Szenenwert[10]; tooltip 0 % = Off 1 - 100 % = Dim level 101 % = Mask; editable
rectangle at (165,255)-(191,281): text "18"; alarm colour if Dali_Config.Kurzadr[18]
rectangle at (190,255)-(231,281): text "%s"; shows DALI_Config.Szenenwert[18]; tooltip 0 % = Off 1 - 100 % = Dim level 101 % = Mask; editable
rectangle at (165,295)-(191,321): text "26"; alarm colour if Dali_Config.Kurzadr[26]
rectangle at (190,295)-(231,321): text "%s"; shows DALI_Config.Szenenwert[26]; tooltip 0 % = Off 1 - 100 % = Dim level 101 % = Mask; editable
rectangle at (165,335)-(191,361): text "34"; alarm colour if Dali_Config.Kurzadr[34]
rectangle at (190,335)-(231,361): text "%s"; shows DALI_Config.Szenenwert[34]; tooltip 0 % = Off 1 - 100 % = Dim level 101 % = Mask; editable
rectangle at (165,375)-(191,401): text "42"; alarm colour if Dali_Config.Kurzadr[42]
rectangle at (190,375)-(231,401): text "%s"; shows DALI_Config.Szenenwert[42]; tooltip 0 % = Off 1 - 100 % = Dim level 101 % = Mask; editable
rectangle at (165,415)-(191,441): text "50"; alarm colour if Dali_Config.Kurzadr[50]
rectangle at (190,415)-(231,441): text "%s"; shows DALI_Config.Szenenwert[50]; tooltip 0 % = Off 1 - 100 % = Dim level 101 % = Mask; editable
rectangle at (165,455)-(191,481): text "58"; alarm colour if Dali_Config.Kurzadr[58]
rectangle at (190,455)-(231,481): text "%s"; shows DALI_Config.Szenenwert[58]; tooltip 0 % = Off 1 - 100 % = Dim level 101 % = Mask; editable
rectangle at (245,175)-(271,201): text "3"; alarm colour if Dali_Config.Kurzadr[3]
rectangle at (270,175)-(311,201): text "%s"; shows DALI_Config.Szenenwert[3]; tooltip 0 % = Off 1 - 100 % = Dim level 101 % = Mask; editable
rectangle at (245,215)-(271,241): text "11"; alarm colour if Dali_Config.Kurzadr[11]
rectangle at (270,215)-(311,241): text "%s"; shows DALI_Config.Szenenwert[11]; tooltip 0 % = Off 1 - 100 % = Dim level 101 % = Mask; editable
rectangle at (245,255)-(271,281): text "19"; alarm colour if Dali_Config.Kurzadr[19]
rectangle at (270,255)-(311,281): text "%s"; shows DALI_Config.Szenenwert[19]; tooltip 0 % = Off 1 - 100 % = Dim level 101 % = Mask; editable
rectangle at (245,295)-(271,321): text "27"; alarm colour if Dali_Config.Kurzadr[27]
rectangle at (270,295)-(311,321): text "%s"; shows DALI_Config.Szenenwert[27]; tooltip 0 % = Off 1 - 100 % = Dim level 101 % = Mask; editable
rectangle at (245,335)-(271,361): text "35"; alarm colour if Dali_Config.Kurzadr[35]
rectangle at (270,335)-(311,361): text "%s"; shows DALI_Config.Szenenwert[35]; tooltip 0 % = Off 1 - 100 % = Dim level 101 % = Mask; editable
rectangle at (245,375)-(271,401): text "43"; alarm colour if Dali_Config.Kurzadr[43]
rectangle at (270,375)-(311,401): text "%s"; shows DALI_Config.Szenenwert[43]; tooltip 0 % = Off 1 - 100 % = Dim level 101 % = Mask; editable
rectangle at (245,415)-(271,441): text "51"; alarm colour if Dali_Config.Kurzadr[51]
rectangle at (270,415)-(311,441): text "%s"; shows DALI_Config.Szenenwert[51]; tooltip 0 % = Off 1 - 100 % = Dim level 101 % = Mask; editable
rectangle at (245,455)-(271,481): text "59"; alarm colour if Dali_Config.Kurzadr[59]
rectangle at (270,455)-(311,481): text "%s"; shows DALI_Config.Szenenwert[59]; tooltip 0 % = Off 1 - 100 % = Dim level 101 % = Mask; editable
rectangle at (325,175)-(351,201): text "4"; alarm colour if Dali_Config.Kurzadr[4]
rectangle at (350,175)-(391,201): text "%s"; shows DALI_Config.Szenenwert[4]; tooltip 0 % = Off 1 - 100 % = Dim level 101 % = Mask; editable
rectangle at (325,215)-(351,241): text "12"; alarm colour if Dali_Config.Kurzadr[12]
rectangle at (350,215)-(391,241): text "%s"; shows DALI_Config.Szenenwert[12]; tooltip 0 % = Off 1 - 100 % = Dim level 101 % = Mask; editable
rectangle at (325,255)-(351,281): text "20"; alarm colour if Dali_Config.Kurzadr[20]
rectangle at (350,255)-(391,281): text "%s"; shows DALI_Config.Szenenwert[20]; tooltip 0 % = Off 1 - 100 % = Dim level 101 % = Mask; editable
rectangle at (325,295)-(351,321): text "28"; alarm colour if Dali_Config.Kurzadr[28]
rectangle at (350,295)-(391,321): text "%s"; shows DALI_Config.Szenenwert[28]; tooltip 0 % = Off 1 - 100 % = Dim level 101 % = Mask; editable
rectangle at (325,335)-(351,361): text "36"; alarm colour if Dali_Config.Kurzadr[36]
rectangle at (350,335)-(391,361): text "%s"; shows DALI_Config.Szenenwert[36]; tooltip 0 % = Off 1 - 100 % = Dim level 101 % = Mask; editable
rectangle at (325,375)-(351,401): text "44"; alarm colour if Dali_Config.Kurzadr[44]
rectangle at (350,375)-(391,401): text "%s"; shows DALI_Config.Szenenwert[44]; tooltip 0 % = Off 1 - 100 % = Dim level 101 % = Mask; editable
rectangle at (325,415)-(351,441): text "52"; alarm colour if Dali_Config.Kurzadr[52]
rectangle at (350,415)-(391,441): text "%s"; shows DALI_Config.Szenenwert[52]; tooltip 0 % = Off 1 - 100 % = Dim level 101 % = Mask; editable
rectangle at (325,455)-(351,481): text "60"; alarm colour if Dali_Config.Kurzadr[60]
rectangle at (350,455)-(391,481): text "%s"; shows DALI_Config.Szenenwert[60]; tooltip 0 % = Off 1 - 100 % = Dim level 101 % = Mask; editable
rectangle at (405,175)-(431,201): text "5"; alarm colour if Dali_Config.Kurzadr[5]
rectangle at (430,175)-(471,201): text "%s"; shows DALI_Config.Szenenwert[5]; tooltip 0 % = Off 1 - 100 % = Dim level 101 % = Mask; editable
rectangle at (405,215)-(431,241): text "13"; alarm colour if Dali_Config.Kurzadr[13]
rectangle at (430,215)-(471,241): text "%s"; shows DALI_Config.Szenenwert[13]; tooltip 0 % = Off 1 - 100 % = Dim level 101 % = Mask; editable
rectangle at (405,255)-(431,281): text "21"; alarm colour if Dali_Config.Kurzadr[21]
rectangle at (430,255)-(471,281): text "%s"; shows DALI_Config.Szenenwert[21]; tooltip 0 % = Off 1 - 100 % = Dim level 101 % = Mask; editable
rectangle at (405,295)-(431,321): text "29"; alarm colour if Dali_Config.Kurzadr[29]
rectangle at (430,295)-(471,321): text "%s"; shows DALI_Config.Szenenwert[29]; tooltip 0 % = Off 1 - 100 % = Dim level 101 % = Mask; editable
rectangle at (405,335)-(431,361): text "37"; alarm colour if Dali_Config.Kurzadr[37]
rectangle at (430,335)-(471,361): text "%s"; shows DALI_Config.Szenenwert[37]; tooltip 0 % = Off 1 - 100 % = Dim level 101 % = Mask; editable
rectangle at (405,375)-(431,401): text "45"; alarm colour if Dali_Config.Kurzadr[45]
rectangle at (430,375)-(471,401): text "%s"; shows DALI_Config.Szenenwert[45]; tooltip 0 % = Off 1 - 100 % = Dim level 101 % = Mask; editable
rectangle at (405,415)-(431,441): text "53"; alarm colour if Dali_Config.Kurzadr[53]
rectangle at (430,415)-(471,441): text "%s"; shows DALI_Config.Szenenwert[53]; tooltip 0 % = Off 1 - 100 % = Dim level 101 % = Mask; editable
rectangle at (405,455)-(431,481): text "61"; alarm colour if Dali_Config.Kurzadr[61]
rectangle at (430,455)-(471,481): text "%s"; shows DALI_Config.Szenenwert[61]; tooltip 0 % = Off 1 - 100 % = Dim level 101 % = Mask; editable
rectangle at (485,175)-(511,201): text "6"; alarm colour if Dali_Config.Kurzadr[6]
rectangle at (510,175)-(551,201): text "%s"; shows DALI_Config.Szenenwert[6]; tooltip 0 % = Off 1 - 100 % = Dim level 101 % = Mask; editable
rectangle at (485,215)-(511,241): text "14"; alarm colour if Dali_Config.Kurzadr[14]
rectangle at (510,215)-(551,241): text "%s"; shows DALI_Config.Szenenwert[14]; tooltip 0 % = Off 1 - 100 % = Dim level 101 % = Mask; editable
rectangle at (485,255)-(511,281): text "22"; alarm colour if Dali_Config.Kurzadr[22]
rectangle at (510,255)-(551,281): text "%s"; shows DALI_Config.Szenenwert[22]; tooltip 0 % = Off 1 - 100 % = Dim level 101 % = Mask; editable
rectangle at (485,295)-(511,321): text "30"; alarm colour if Dali_Config.Kurzadr[30]
rectangle at (510,295)-(551,321): text "%s"; shows DALI_Config.Szenenwert[30]; tooltip 0 % = Off 1 - 100 % = Dim level 101 % = Mask; editable
rectangle at (485,335)-(511,361): text "38"; alarm colour if Dali_Config.Kurzadr[38]
rectangle at (510,335)-(551,361): text "%s"; shows DALI_Config.Szenenwert[38]; tooltip 0 % = Off 1 - 100 % = Dim level 101 % = Mask; editable
rectangle at (485,375)-(511,401): text "46"; alarm colour if Dali_Config.Kurzadr[46]
rectangle at (510,375)-(551,401): text "%s"; shows DALI_Config.Szenenwert[46]; tooltip 0 % = Off 1 - 100 % = Dim level 101 % = Mask; editable
rectangle at (485,415)-(511,441): text "54"; alarm colour if Dali_Config.Kurzadr[54]
rectangle at (510,415)-(551,441): text "%s"; shows DALI_Config.Szenenwert[54]; tooltip 0 % = Off 1 - 100 % = Dim level 101 % = Mask; editable
rectangle at (485,455)-(511,481): text "62"; alarm colour if Dali_Config.Kurzadr[62]
rectangle at (510,455)-(551,481): text "%s"; shows DALI_Config.Szenenwert[62]; tooltip 0 % = Off 1 - 100 % = Dim level 101 % = Mask; editable
rectangle at (565,175)-(591,201): text "7"; alarm colour if Dali_Config.Kurzadr[7]
rectangle at (590,175)-(631,201): text "%s"; shows DALI_Config.Szenenwert[7]; tooltip 0 % = Off 1 - 100 % = Dim level 101 % = Mask; editable
rectangle at (565,215)-(591,241): text "15"; alarm colour if Dali_Config.Kurzadr[15]
rectangle at (590,215)-(631,241): text "%s"; shows DALI_Config.Szenenwert[15]; tooltip 0 % = Off 1 - 100 % = Dim level 101 % = Mask; editable
rectangle at (565,255)-(591,281): text "23"; alarm colour if Dali_Config.Kurzadr[23]
rectangle at (590,255)-(631,281): text "%s"; shows DALI_Config.Szenenwert[23]; tooltip 0 % = Off 1 - 100 % = Dim level 101 % = Mask; editable
rectangle at (565,295)-(591,321): text "31"; alarm colour if Dali_Config.Kurzadr[31]
rectangle at (590,295)-(631,321): text "%s"; shows DALI_Config.Szenenwert[31]; tooltip 0 % = Off 1 - 100 % = Dim level 101 % = Mask; editable
rectangle at (565,335)-(591,361): text "39"; alarm colour if Dali_Config.Kurzadr[39]
rectangle at (590,335)-(631,361): text "%s"; shows DALI_Config.Szenenwert[39]; tooltip 0 % = Off 1 - 100 % = Dim level 101 % = Mask; editable
rectangle at (565,375)-(591,401): text "47"; alarm colour if Dali_Config.Kurzadr[47]
rectangle at (590,375)-(631,401): text "%s"; shows DALI_Config.Szenenwert[47]; tooltip 0 % = Off 1 - 100 % = Dim level 101 % = Mask; editable
rectangle at (565,415)-(591,441): text "55"; alarm colour if Dali_Config.Kurzadr[55]
rectangle at (590,415)-(631,441): text "%s"; shows DALI_Config.Szenenwert[55]; tooltip 0 % = Off 1 - 100 % = Dim level 101 % = Mask; editable
rectangle at (565,455)-(591,481): text "63"; alarm colour if Dali_Config.Kurzadr[63]
rectangle at (590,455)-(631,481): text "%s"; shows DALI_Config.Szenenwert[63]; tooltip 0 % = Off 1 - 100 % = Dim level 101 % = Mask; editable
rectangle at (645,175)-(671,201): text "8"; alarm colour if Dali_Config.Kurzadr[8]
rectangle at (670,175)-(711,201): text "%s"; shows DALI_Config.Szenenwert[8]; tooltip 0 % = Off 1 - 100 % = Dim level 101 % = Mask; editable
rectangle at (645,215)-(671,241): text "16"; alarm colour if Dali_Config.Kurzadr[16]
rectangle at (670,215)-(711,241): text "%s"; shows DALI_Config.Szenenwert[16]; tooltip 0 % = Off 1 - 100 % = Dim level 101 % = Mask; editable
rectangle at (645,255)-(671,281): text "24"; alarm colour if Dali_Config.Kurzadr[24]
rectangle at (670,255)-(711,281): text "%s"; shows DALI_Config.Szenenwert[24]; tooltip 0 % = Off 1 - 100 % = Dim level 101 % = Mask; editable
rectangle at (645,295)-(671,321): text "32"; alarm colour if Dali_Config.Kurzadr[32]
rectangle at (670,295)-(711,321): text "%s"; shows DALI_Config.Szenenwert[32]; tooltip 0 % = Off 1 - 100 % = Dim level 101 % = Mask; editable
rectangle at (645,335)-(671,361): text "40"; alarm colour if Dali_Config.Kurzadr[40]
rectangle at (670,335)-(711,361): text "%s"; shows DALI_Config.Szenenwert[40]; tooltip 0 % = Off 1 - 100 % = Dim level 101 % = Mask; editable
rectangle at (645,375)-(671,401): text "48"; alarm colour if Dali_Config.Kurzadr[48]
rectangle at (670,375)-(711,401): text "%s"; shows DALI_Config.Szenenwert[48]; tooltip 0 % = Off 1 - 100 % = Dim level 101 % = Mask; editable
rectangle at (645,415)-(671,441): text "56"; alarm colour if Dali_Config.Kurzadr[56]
rectangle at (670,415)-(711,441): text "%s"; shows DALI_Config.Szenenwert[56]; tooltip 0 % = Off 1 - 100 % = Dim level 101 % = Mask; editable
rectangle at (645,455)-(671,481): text "64"; alarm colour if Dali_Config.Kurzadr[64]
rectangle at (670,455)-(711,481): text "%s"; shows DALI_Config.Szenenwert[64]; tooltip 0 % = Off 1 - 100 % = Dim level 101 % = Mask; editable
rectangle at (165,115)-(281,151): text "Scene:"
rectangle at (285,115)-(321,151): text "%s"; shows DALI_Config.Szene; tooltip Select scene 1 - 16; editable
rectangle at (110,505)-(261,526): text "Short address available"
rectangle at (105,535)-(291,556): text "Short address not assigned"
rectangle at (51,111)-(742,498): text "Please wait!"; invisible if NOT DALI_Config.Unsichtbar
4 more shapes without text or variables
*)

